LIN {X 0,Y 316.561,Z 503.563,A -85,B 0,C 180,E1 -16116.935,E2 -16116.935} C_VEL
LIN {X 0,Y 317.604,Z 489.042,A -85,B 0,C 180,E1 -16117.711,E2 -16117.711} C_VEL
LIN {X 0,Y 318.34,Z 474.612,A -85,B 0,C 180,E1 -16118.212,E2 -16118.212} C_VEL
LIN {X 0,Y 320.9,Z 379.662,A -85,B 0,C 180,E1 -16120.351,E2 -16120.351} C_VEL
LIN {X 0,Y 312.797,Z 358.488,A -85,B 0,C 180,E1 -16121.547,E2 -16121.547} C_VEL
LIN {X 0,Y 305.815,Z 342.039,A -85,B 0,C 180,E1 -16122.612,E2 -16122.612} C_VEL
LIN {X 0,Y 305.593,Z 341.045,A -85,B 0,C 180,E1 -16122.959,E2 -16122.959} C_VEL
LIN {X 0,Y 305.551,Z 341.05,A -85,B 0,C 180,E1 -16126.023,E2 -16126.023} C_VEL
LIN {X 0,Y 305.541,Z 341.055,A -85,B 0,C 180,E1 -16129.428,E2 -16129.428} C_VEL
LIN {X 0,Y 305.486,Z 341.061,A -85,B 0,C 180,E1 -16133.04,E2 -16133.04} C_VEL
LIN {X 0,Y 305.466,Z 341.058,A -85,B 0,C 180,E1 -16136.197,E2 -16136.197} C_VEL
LIN {X 0,Y 305.433,Z 341.065,A -85,B 0,C 180,E1 -16139.03,E2 -16139.03} C_VEL
LIN {X 0,Y 305.434,Z 341.061,A -85,B 0,C 180,E1 -16141.954,E2 -16141.954} C_VEL
LIN {X 0,Y 305.46,Z 341.058,A -85,B 0,C 180,E1 -16145.115,E2 -16145.115} C_VEL
LIN {X 0,Y 305.432,Z 341.061,A -85,B 0,C 180,E1 -16148.526,E2 -16148.526} C_VEL
LIN {X 0,Y 305.391,Z 341.064,A -85,B 0,C 180,E1 -16149.611,E2 -16149.611} C_VEL
LIN {X 0,Y 304.744,Z 341.152,A -85,B 0,C 180,E1 -16150.712,E2 -16150.712} C_VEL
LIN {X 0,Y 301.909,Z 341.502,A -85,B 0,C 180,E1 -16152.504,E2 -16152.504} C_VEL
LIN {X 0,Y 299.483,Z 341.8,A -85,B 0,C 180,E1 -16153.957,E2 -16153.957} C_VEL
LIN {X 0,Y 298.425,Z 341.93,A -85,B 0,C 180,E1 -16155.083,E2 -16155.083} C_VEL
LIN {X 0,Y 298.331,Z 341.939,A -85,B 0,C 180,E1 -16155.464,E2 -16155.464} C_VEL
LIN {X 0,Y 298.348,Z 341.946,A -85,B 0,C 180,E1 -16158.922,E2 -16158.922} C_VEL
LIN {X 0,Y 298.427,Z 341.922,A -85,B 0,C 180,E1 -16163.199,E2 -16163.199} C_VEL
LIN {X 0,Y 298.394,Z 341.937,A -85,B 0,C 180,E1 -16167.2,E2 -16167.2} C_VEL
LIN {X 0,Y 298.366,Z 341.944,A -85,B 0,C 180,E1 -16170.639,E2 -16170.639} C_VEL
LIN {X 0,Y 298.414,Z 341.937,A -85,B 0,C 180,E1 -16174.918,E2 -16174.918} C_VEL
LIN {X 0,Y 298.394,Z 341.938,A -85,B 0,C 180,E1 -16177.862,E2 -16177.862} C_VEL
LIN {X 0,Y 298.464,Z 341.931,A -85,B 0,C 180,E1 -16180.752,E2 -16180.752} C_VEL
LIN {X 0,Y 298.513,Z 341.917,A -85,B 0,C 180,E1 -16184.991,E2 -16184.991} C_VEL
LIN {X 0,Y 298.585,Z 341.905,A -85,B 0,C 180,E1 -16189.147,E2 -16189.147} C_VEL
LIN {X 0,Y 298.702,Z 341.9,A -85,B 0,C 180,E1 -16191.885,E2 -16191.885} C_VEL
LIN {X 0,Y 298.639,Z 341.908,A -85,B 0,C 180,E1 -16194.599,E2 -16194.599} C_VEL
LIN {X 0,Y 298.92,Z 341.861,A -85,B 0,C 180,E1 -16198.653,E2 -16198.653} C_VEL
LIN {X 0,Y 298.92,Z 341.864,A -85,B 0,C 180,E1 -16201.348,E2 -16201.348} C_VEL
LIN {X 0,Y 298.752,Z 341.893,A -85,B 0,C 180,E1 -16206.755,E2 -16206.755} C_VEL
LIN {X 0,Y 298.63,Z 341.909,A -85,B 0,C 180,E1 -16209.483,E2 -16209.483} C_VEL
LIN {X 0,Y 298.557,Z 341.92,A -85,B 0,C 180,E1 -16213.616,E2 -16213.616} C_VEL
LIN {X 0,Y 298.554,Z 341.919,A -85,B 0,C 180,E1 -16216.409,E2 -16216.409} C_VEL
LIN {X 0,Y 298.516,Z 341.923,A -85,B 0,C 180,E1 -16219.655,E2 -16219.655} C_VEL
LIN {X 0,Y 298.463,Z 341.932,A -85,B 0,C 180,E1 -16223.598,E2 -16223.598} C_VEL
LIN {X 0,Y 298.492,Z 341.925,A -85,B 0,C 180,E1 -16226.575,E2 -16226.575} C_VEL
LIN {X 0,Y 298.421,Z 341.936,A -85,B 0,C 180,E1 -16229.641,E2 -16229.641} C_VEL
LIN {X 0,Y 298.4,Z 341.938,A -85,B 0,C 180,E1 -16232.8,E2 -16232.8} C_VEL
LIN {X 0,Y 298.45,Z 341.932,A -85,B 0,C 180,E1 -16236.807,E2 -16236.807} C_VEL
LIN {X 0,Y 298.393,Z 341.943,A -85,B 0,C 180,E1 -16241.088,E2 -16241.088} C_VEL
LIN {X 0,Y 298.393,Z 341.942,A -85,B 0,C 180,E1 -16245.041,E2 -16245.041} C_VEL
LIN {X 0,Y 298.393,Z 341.944,A -85,B 0,C 180,E1 -16248.912,E2 -16248.912} C_VEL
LIN {X 0,Y 298.451,Z 341.937,A -85,B 0,C 180,E1 -16253.192,E2 -16253.192} C_VEL
LIN {X 0,Y 298.484,Z 342.254,A -85,B 0,C 180,E1 -16253.458,E2 -16253.458} C_VEL
LIN {X 0,Y 301.039,Z 352.934,A -85,B 0,C 180,E1 -16256.6,E2 -16256.6} C_VEL
LIN {X 0,Y 303.03,Z 362.138,A -85,B 0,C 180,E1 -16259.159,E2 -16259.159} C_VEL
LIN {X 0,Y 308.535,Z 376.907,A -85,B 0,C 180,E1 -16260.032,E2 -16260.032} C_VEL
LIN {X 0,Y 313.753,Z 411.636,A -85,B 0,C 180,E1 -16261.349,E2 -16261.349} C_VEL
LIN {X 0,Y 311.27,Z 499.633,A -85,B 0,C 180,E1 -16263.381,E2 -16263.381} C_VEL
LIN {X 0,Y 310.406,Z 513.885,A -85,B 0,C 180,E1 -16263.934,E2 -16263.934} C_VEL
LIN {X 0,Y 309.038,Z 528.229,A -85,B 0,C 180,E1 -16264.759,E2 -16264.759} C_VEL
LIN {X 0,Y 307.585,Z 540.599,A -85,B 0,C 180,E1 -16265.714,E2 -16265.714} C_VEL
LIN {X 0,Y 305.986,Z 553.621,A -85,B 0,C 180,E1 -16267.016,E2 -16267.016} C_VEL
LIN {X 0,Y 304.401,Z 564.227,A -85,B 0,C 180,E1 -16268.32,E2 -16268.32} C_VEL
LIN {X 0,Y 302.566,Z 575.211,A -85,B 0,C 180,E1 -16269.963,E2 -16269.963} C_VEL
LIN {X 0,Y 300.847,Z 586.07,A -85,B 0,C 180,E1 -16271.968,E2 -16271.968} C_VEL
LIN {X 0,Y 299.37,Z 595.713,A -85,B 0,C 180,E1 -16274.162,E2 -16274.162} C_VEL
LIN {X 0,Y 298.435,Z 602.452,A -85,B 0,C 180,E1 -16276.031,E2 -16276.031} C_VEL
LIN {X 0,Y 297.468,Z 609.537,A -85,B 0,C 180,E1 -16278.414,E2 -16278.414} C_VEL
LIN {X 0,Y 296.971,Z 614.436,A -85,B 0,C 180,E1 -16280.463,E2 -16280.463} C_VEL
LIN {X 0,Y 296.656,Z 619.479,A -85,B 0,C 180,E1 -16283.196,E2 -16283.196} C_VEL
LIN {X 0,Y 296.569,Z 622.979,A -85,B 0,C 180,E1 -16285.922,E2 -16285.922} C_VEL
LIN {X 0,Y 296.561,Z 625.044,A -85,B 0,C 180,E1 -16288.641,E2 -16288.641} C_VEL
LIN {X 0,Y 296.583,Z 625.56,A -85,B 0,C 180,E1 -16289.999,E2 -16289.999} C_VEL
LIN {X 0,Y 296.544,Z 625.573,A -85,B 0,C 180,E1 -16292.716,E2 -16292.716} C_VEL
LIN {X 0,Y 296.546,Z 624.19,A -85,B 0,C 180,E1 -16295.507,E2 -16295.507} C_VEL
LIN {X 0,Y 296.813,Z 621.558,A -85,B 0,C 180,E1 -16298.166,E2 -16298.166} C_VEL
LIN {X 0,Y 297.411,Z 617.457,A -85,B 0,C 180,E1 -16300.896,E2 -16300.896} C_VEL
LIN {X 0,Y 298.62,Z 611.832,A -85,B 0,C 180,E1 -16303.611,E2 -16303.611} C_VEL
LIN {X 0,Y 300.197,Z 604.52,A -85,B 0,C 180,E1 -16306.315,E2 -16306.315} C_VEL
LIN {X 0,Y 302.199,Z 596.494,A -85,B 0,C 180,E1 -16308.648,E2 -16308.648} C_VEL
LIN {X 0,Y 304.312,Z 588.131,A -85,B 0,C 180,E1 -16310.62,E2 -16310.62} C_VEL
LIN {X 0,Y 306.857,Z 578.101,A -85,B 0,C 180,E1 -16312.557,E2 -16312.557} C_VEL
LIN {X 0,Y 309.221,Z 568.042,A -85,B 0,C 180,E1 -16314.147,E2 -16314.147} C_VEL
LIN {X 0,Y 311.767,Z 555.927,A -85,B 0,C 180,E1 -16315.716,E2 -16315.716} C_VEL
LIN {X 0,Y 314.08,Z 543.986,A -85,B 0,C 180,E1 -16316.943,E2 -16316.943} C_VEL
LIN {X 0,Y 316.223,Z 530.835,A -85,B 0,C 180,E1 -16318,E2 -16318} C_VEL
LIN {X 0,Y 318.041,Z 517.262,A -85,B 0,C 180,E1 -16318.815,E2 -16318.815} C_VEL
LIN {X 0,Y 319.406,Z 503.345,A -85,B 0,C 180,E1 -16319.401,E2 -16319.401} C_VEL
LIN {X 0,Y 320.305,Z 484.536,A -85,B 0,C 180,E1 -16319.898,E2 -16319.898} C_VEL
LIN {X 0,Y 322.883,Z 413.283,A -85,B 0,C 180,E1 -16321.53,E2 -16321.53} C_VEL
LIN {X 0,Y 320.316,Z 397.518,A -85,B 0,C 180,E1 -16322.31,E2 -16322.31} C_VEL
LIN {X 0,Y 318.901,Z 390.848,A -85,B 0,C 180,E1 -16322.692,E2 -16322.692} C_VEL
LIN {X 0,Y 312.51,Z 377.162,A -85,B 0,C 180,E1 -16324.007,E2 -16324.007} C_VEL
LIN {X 0,Y 306.262,Z 365.122,A -85,B 0,C 180,E1 -16325.339,E2 -16325.339} C_VEL
LIN {X 0,Y 303.755,Z 360.397,A -85,B 0,C 180,E1 -16325.923,E2 -16325.923} C_VEL
LIN {X 0,Y 300.958,Z 350.238,A -85,B 0,C 180,E1 -16329.59,E2 -16329.59} C_VEL
LIN {X 0,Y 298.426,Z 341.929,A -85,B 0,C 180,E1 -16332.924,E2 -16332.924} C_VEL
LIN {X 0,Y 298.398,Z 341.929,A -85,B 0,C 180,E1 -16336.919,E2 -16336.919} C_VEL
LIN {X 0,Y 298.41,Z 341.919,A -85,B 0,C 180,E1 -16341.002,E2 -16341.002} C_VEL
LIN {X 0,Y 298.426,Z 341.933,A -85,B 0,C 180,E1 -16343.931,E2 -16343.931} C_VEL
LIN {X 0,Y 298.39,Z 341.937,A -85,B 0,C 180,E1 -16347.982,E2 -16347.982} C_VEL
LIN {X 0,Y 298.458,Z 341.933,A -85,B 0,C 180,E1 -16351.903,E2 -16351.903} C_VEL
LIN {X 0,Y 298.479,Z 341.931,A -85,B 0,C 180,E1 -16354.923,E2 -16354.923} C_VEL
LIN {X 0,Y 298.443,Z 341.935,A -85,B 0,C 180,E1 -16359.314,E2 -16359.314} C_VEL
LIN {X 0,Y 298.531,Z 341.92,A -85,B 0,C 180,E1 -16362.179,E2 -16362.179} C_VEL
LIN {X 0,Y 298.586,Z 341.906,A -85,B 0,C 180,E1 -16364.994,E2 -16364.994} C_VEL
LIN {X 0,Y 298.586,Z 341.905,A -85,B 0,C 180,E1 -16369.146,E2 -16369.146} C_VEL
LIN {X 0,Y 298.75,Z 341.892,A -85,B 0,C 180,E1 -16371.885,E2 -16371.885} C_VEL
LIN {X 0,Y 298.643,Z 341.909,A -85,B 0,C 180,E1 -16374.598,E2 -16374.598} C_VEL
LIN {X 0,Y 298.906,Z 341.876,A -85,B 0,C 180,E1 -16378.652,E2 -16378.652} C_VEL
LIN {X 0,Y 298.895,Z 341.869,A -85,B 0,C 180,E1 -16381.347,E2 -16381.347} C_VEL
LIN {X 0,Y 298.693,Z 341.9,A -85,B 0,C 180,E1 -16386.513,E2 -16386.513} C_VEL
LIN {X 0,Y 298.616,Z 341.905,A -85,B 0,C 180,E1 -16389.482,E2 -16389.482} C_VEL
LIN {X 0,Y 298.534,Z 341.919,A -85,B 0,C 180,E1 -16393.616,E2 -16393.616} C_VEL
LIN {X 0,Y 298.474,Z 341.923,A -85,B 0,C 180,E1 -16396.412,E2 -16396.412} C_VEL
LIN {X 0,Y 298.451,Z 341.929,A -85,B 0,C 180,E1 -16399.627,E2 -16399.627} C_VEL
LIN {X 0,Y 298.411,Z 341.941,A -85,B 0,C 180,E1 -16403.601,E2 -16403.601} C_VEL
LIN {X 0,Y 298.399,Z 341.943,A -85,B 0,C 180,E1 -16406.582,E2 -16406.582} C_VEL
LIN {X 0,Y 298.385,Z 341.93,A -85,B 0,C 180,E1 -16409.644,E2 -16409.644} C_VEL
LIN {X 0,Y 298.384,Z 341.932,A -85,B 0,C 180,E1 -16412.801,E2 -16412.801} C_VEL
LIN {X 0,Y 298.448,Z 342.109,A -85,B 0,C 180,E1 -16414.496,E2 -16414.496} C_VEL
LIN {X 0,Y 299.073,Z 344.176,A -85,B 0,C 180,E1 -16415.356,E2 -16415.356} C_VEL
LIN {X 0,Y 301.615,Z 348.304,A -85,B 0,C 180,E1 -16415.931,E2 -16415.931} C_VEL
LIN {X 0,Y 309.75,Z 361.63,A -85,B 0,C 180,E1 -16417.672,E2 -16417.672} C_VEL
LIN {X 0,Y 318.436,Z 377.963,A -85,B 0,C 180,E1 -16419.442,E2 -16419.442} C_VEL
LIN {X 0,Y 323.82,Z 389.532,A -85,B 0,C 180,E1 -16420.501,E2 -16420.501} C_VEL
LIN {X 0,Y 320.298,Z 479.035,A -85,B 0,C 180,E1 -16422.55,E2 -16422.55} C_VEL
LIN {X 0,Y 319.269,Z 493.289,A -85,B 0,C 180,E1 -16423.111,E2 -16423.111} C_VEL
LIN {X 0,Y 317.836,Z 506.14,A -85,B 0,C 180,E1 -16423.832,E2 -16423.832} C_VEL
LIN {X 0,Y 316.098,Z 519.195,A -85,B 0,C 180,E1 -16424.828,E2 -16424.828} C_VEL
LIN {X 0,Y 313.944,Z 531.813,A -85,B 0,C 180,E1 -16426.057,E2 -16426.057} C_VEL
LIN {X 0,Y 311.486,Z 544.174,A -85,B 0,C 180,E1 -16427.577,E2 -16427.577} C_VEL
LIN {X 0,Y 308.852,Z 555.794,A -85,B 0,C 180,E1 -16429.357,E2 -16429.357} C_VEL
LIN {X 0,Y 306.313,Z 566.384,A -85,B 0,C 180,E1 -16431.383,E2 -16431.383} C_VEL
LIN {X 0,Y 304.021,Z 575.007,A -85,B 0,C 180,E1 -16433.415,E2 -16433.415} C_VEL
LIN {X 0,Y 301.963,Z 582.651,A -85,B 0,C 180,E1 -16435.641,E2 -16435.641} C_VEL
LIN {X 0,Y 300.116,Z 589.603,A -85,B 0,C 180,E1 -16438.206,E2 -16438.206} C_VEL
LIN {X 0,Y 298.826,Z 594.434,A -85,B 0,C 180,E1 -16440.48,E2 -16440.48} C_VEL
LIN {X 0,Y 297.685,Z 598.912,A -85,B 0,C 180,E1 -16443.35,E2 -16443.35} C_VEL
LIN {X 0,Y 296.885,Z 601.861,A -85,B 0,C 180,E1 -16446.271,E2 -16446.271} C_VEL
LIN {X 0,Y 296.685,Z 602.753,A -85,B 0,C 180,E1 -16447.729,E2 -16447.729} C_VEL
LIN {X 0,Y 296.391,Z 603.41,A -85,B 0,C 180,E1 -16450.613,E2 -16450.613} C_VEL
LIN {X 0,Y 296.359,Z 603.175,A -85,B 0,C 180,E1 -16452.045,E2 -16452.045} C_VEL
LIN {X 0,Y 296.359,Z 601.642,A -85,B 0,C 180,E1 -16454.88,E2 -16454.88} C_VEL
LIN {X 0,Y 296.559,Z 600.305,A -85,B 0,C 180,E1 -16456.319,E2 -16456.319} C_VEL
LIN {X 0,Y 296.964,Z 596.634,A -85,B 0,C 180,E1 -16459.088,E2 -16459.088} C_VEL
LIN {X 0,Y 297.636,Z 591.401,A -85,B 0,C 180,E1 -16461.856,E2 -16461.856} C_VEL
LIN {X 0,Y 298.375,Z 586.318,A -85,B 0,C 180,E1 -16463.917,E2 -16463.917} C_VEL
LIN {X 0,Y 299.441,Z 579.063,A -85,B 0,C 180,E1 -16466.301,E2 -16466.301} C_VEL
LIN {X 0,Y 300.707,Z 571.447,A -85,B 0,C 180,E1 -16468.327,E2 -16468.327} C_VEL
LIN {X 0,Y 302.204,Z 562.576,A -85,B 0,C 180,E1 -16470.278,E2 -16470.278} C_VEL
LIN {X 0,Y 303.619,Z 553.219,A -85,B 0,C 180,E1 -16471.991,E2 -16471.991} C_VEL
LIN {X 0,Y 305.369,Z 542.327,A -85,B 0,C 180,E1 -16473.63,E2 -16473.63} C_VEL
LIN {X 0,Y 307.014,Z 530.442,A -85,B 0,C 180,E1 -16475.09,E2 -16475.09} C_VEL
LIN {X 0,Y 308.604,Z 517.319,A -85,B 0,C 180,E1 -16476.375,E2 -16476.375} C_VEL
LIN {X 0,Y 309.972,Z 503.451,A -85,B 0,C 180,E1 -16477.41,E2 -16477.41} C_VEL
LIN {X 0,Y 311.041,Z 488.778,A -85,B 0,C 180,E1 -16478.201,E2 -16478.201} C_VEL
LIN {X 0,Y 311.728,Z 475.513,A -85,B 0,C 180,E1 -16478.673,E2 -16478.673} C_VEL
LIN {X 0,Y 314.484,Z 381.922,A -85,B 0,C 180,E1 -16480.813,E2 -16480.813} C_VEL
LIN {X 0,Y 308.384,Z 365.374,A -85,B 0,C 180,E1 -16481.754,E2 -16481.754} C_VEL
LIN {X 0,Y 299.779,Z 345.144,A -85,B 0,C 180,E1 -16483.072,E2 -16483.072} C_VEL
LIN {X 0,Y 298.606,Z 342.346,A -85,B 0,C 180,E1 -16483.268,E2 -16483.268} C_VEL
LIN {X 0,Y 298.552,Z 341.923,A -85,B 0,C 180,E1 -16483.443,E2 -16483.443} C_VEL
LIN {X 0,Y 298.485,Z 341.931,A -85,B 0,C 180,E1 -16486.413,E2 -16486.413} C_VEL
LIN {X 0,Y 298.482,Z 341.933,A -85,B 0,C 180,E1 -16489.64,E2 -16489.64} C_VEL
LIN {X 0,Y 298.419,Z 341.938,A -85,B 0,C 180,E1 -16493.602,E2 -16493.602} C_VEL
LIN {X 0,Y 298.406,Z 341.939,A -85,B 0,C 180,E1 -16496.583,E2 -16496.583} C_VEL
LIN {X 0,Y 298.36,Z 341.944,A -85,B 0,C 180,E1 -16499.649,E2 -16499.649} C_VEL
LIN {X 0,Y 298.391,Z 341.942,A -85,B 0,C 180,E1 -16502.802,E2 -16502.802} C_VEL
LIN {X 0,Y 298.427,Z 341.931,A -85,B 0,C 180,E1 -16506.803,E2 -16506.803} C_VEL
LIN {X 0,Y 298.365,Z 341.942,A -85,B 0,C 180,E1 -16509.591,E2 -16509.591} C_VEL
LIN {X 0,Y 298.369,Z 341.936,A -85,B 0,C 180,E1 -16513.098,E2 -16513.098} C_VEL
LIN {X 0,Y 298.331,Z 341.939,A -85,B 0,C 180,E1 -16515.464,E2 -16515.464} C_VEL
LIN {X 0,Y 297.645,Z 342.031,A -85,B 0,C 180,E1 -16516.592,E2 -16516.592} C_VEL
LIN {X 0,Y 294.807,Z 342.387,A -85,B 0,C 180,E1 -16518.429,E2 -16518.429} C_VEL
LIN {X 0,Y 292.411,Z 342.685,A -85,B 0,C 180,E1 -16519.919,E2 -16519.919} C_VEL
LIN {X 0,Y 291.383,Z 342.808,A -85,B 0,C 180,E1 -16521.073,E2 -16521.073} C_VEL
LIN {X 0,Y 291.298,Z 342.815,A -85,B 0,C 180,E1 -16521.463,E2 -16521.463} C_VEL
LIN {X 0,Y 291.356,Z 342.804,A -85,B 0,C 180,E1 -16524.626,E2 -16524.626} C_VEL
LIN {X 0,Y 291.367,Z 342.812,A -85,B 0,C 180,E1 -16527.951,E2 -16527.951} C_VEL
LIN {X 0,Y 291.317,Z 342.818,A -85,B 0,C 180,E1 -16531.152,E2 -16531.152} C_VEL
LIN {X 0,Y 291.344,Z 342.819,A -85,B 0,C 180,E1 -16534.266,E2 -16534.266} C_VEL
LIN {X 0,Y 291.352,Z 342.813,A -85,B 0,C 180,E1 -16537.298,E2 -16537.298} C_VEL
LIN {X 0,Y 291.389,Z 342.813,A -85,B 0,C 180,E1 -16540.266,E2 -16540.266} C_VEL
LIN {X 0,Y 291.477,Z 342.794,A -85,B 0,C 180,E1 -16544.683,E2 -16544.683} C_VEL
LIN {X 0,Y 291.531,Z 342.784,A -85,B 0,C 180,E1 -16548.881,E2 -16548.881} C_VEL
LIN {X 0,Y 291.655,Z 342.776,A -85,B 0,C 180,E1 -16551.687,E2 -16551.687} C_VEL
LIN {X 0,Y 291.608,Z 342.784,A -85,B 0,C 180,E1 -16554.468,E2 -16554.468} C_VEL
LIN {X 0,Y 291.886,Z 342.735,A -85,B 0,C 180,E1 -16558.621,E2 -16558.621} C_VEL
LIN {X 0,Y 291.886,Z 342.739,A -85,B 0,C 180,E1 -16561.38,E2 -16561.38} C_VEL
LIN {X 0,Y 291.704,Z 342.771,A -85,B 0,C 180,E1 -16566.919,E2 -16566.919} C_VEL
LIN {X 0,Y 291.573,Z 342.789,A -85,B 0,C 180,E1 -16569.714,E2 -16569.714} C_VEL
LIN {X 0,Y 291.527,Z 342.795,A -85,B 0,C 180,E1 -16573.95,E2 -16573.95} C_VEL
LIN {X 0,Y 291.492,Z 342.798,A -85,B 0,C 180,E1 -16576.818,E2 -16576.818} C_VEL
LIN {X 0,Y 291.456,Z 342.802,A -85,B 0,C 180,E1 -16579.875,E2 -16579.875} C_VEL
LIN {X 0,Y 291.405,Z 342.806,A -85,B 0,C 180,E1 -16584.205,E2 -16584.205} C_VEL
LIN {X 0,Y 291.425,Z 342.808,A -85,B 0,C 180,E1 -16587.272,E2 -16587.272} C_VEL
LIN {X 0,Y 291.339,Z 342.816,A -85,B 0,C 180,E1 -16590.437,E2 -16590.437} C_VEL
LIN {X 0,Y 291.349,Z 342.818,A -85,B 0,C 180,E1 -16593.698,E2 -16593.698} C_VEL
LIN {X 0,Y 291.378,Z 342.811,A -85,B 0,C 180,E1 -16597.253,E2 -16597.253} C_VEL
LIN {X 0,Y 291.338,Z 342.819,A -85,B 0,C 180,E1 -16600.642,E2 -16600.642} C_VEL
LIN {X 0,Y 291.319,Z 342.82,A -85,B 0,C 180,E1 -16604.397,E2 -16604.397} C_VEL
LIN {X 0,Y 291.332,Z 342.821,A -85,B 0,C 180,E1 -16608.404,E2 -16608.404} C_VEL
LIN {X 0,Y 291.358,Z 342.823,A -85,B 0,C 180,E1 -16611.158,E2 -16611.158} C_VEL
LIN {X 0,Y 291.416,Z 342.879,A -85,B 0,C 180,E1 -16612.864,E2 -16612.864} C_VEL
LIN {X 0,Y 294.4,Z 355.607,A -85,B 0,C 180,E1 -16616.696,E2 -16616.696} C_VEL
LIN {X 0,Y 295.8,Z 362.018,A -85,B 0,C 180,E1 -16618.485,E2 -16618.485} C_VEL
LIN {X 0,Y 302.3,Z 379.135,A -85,B 0,C 180,E1 -16619.54,E2 -16619.54} C_VEL
LIN {X 0,Y 307.271,Z 412.118,A -85,B 0,C 180,E1 -16620.83,E2 -16620.83} C_VEL
LIN {X 0,Y 304.68,Z 499.831,A -85,B 0,C 180,E1 -16622.897,E2 -16622.897} C_VEL
LIN {X 0,Y 303.777,Z 513.874,A -85,B 0,C 180,E1 -16623.46,E2 -16623.46} C_VEL
LIN {X 0,Y 302.45,Z 527.587,A -85,B 0,C 180,E1 -16624.262,E2 -16624.262} C_VEL
LIN {X 0,Y 300.833,Z 540.883,A -85,B 0,C 180,E1 -16625.311,E2 -16625.311} C_VEL
LIN {X 0,Y 299.184,Z 553.839,A -85,B 0,C 180,E1 -16626.645,E2 -16626.645} C_VEL
LIN {X 0,Y 297.548,Z 564.359,A -85,B 0,C 180,E1 -16627.977,E2 -16627.977} C_VEL
LIN {X 0,Y 295.81,Z 574.283,A -85,B 0,C 180,E1 -16629.485,E2 -16629.485} C_VEL
LIN {X 0,Y 294.309,Z 583.605,A -85,B 0,C 180,E1 -16631.192,E2 -16631.192} C_VEL
LIN {X 0,Y 292.8,Z 592.929,A -85,B 0,C 180,E1 -16633.259,E2 -16633.259} C_VEL
LIN {X 0,Y 291.727,Z 600.692,A -85,B 0,C 180,E1 -16635.346,E2 -16635.346} C_VEL
LIN {X 0,Y 290.735,Z 607.131,A -85,B 0,C 180,E1 -16637.433,E2 -16637.433} C_VEL
LIN {X 0,Y 290.044,Z 612.404,A -85,B 0,C 180,E1 -16639.528,E2 -16639.528} C_VEL
LIN {X 0,Y 289.648,Z 617.954,A -85,B 0,C 180,E1 -16642.33,E2 -16642.33} C_VEL
LIN {X 0,Y 289.482,Z 621.101,A -85,B 0,C 180,E1 -16644.5,E2 -16644.5} C_VEL
LIN {X 0,Y 289.496,Z 623.832,A -85,B 0,C 180,E1 -16647.216,E2 -16647.216} C_VEL
LIN {X 0,Y 289.498,Z 625.253,A -85,B 0,C 180,E1 -16649.999,E2 -16649.999} C_VEL
LIN {X 0,Y 289.469,Z 625.316,A -85,B 0,C 180,E1 -16652.782,E2 -16652.782} C_VEL
LIN {X 0,Y 289.477,Z 624.043,A -85,B 0,C 180,E1 -16655.572,E2 -16655.572} C_VEL
LIN {X 0,Y 289.746,Z 621.425,A -85,B 0,C 180,E1 -16658.367,E2 -16658.367} C_VEL
LIN {X 0,Y 290.377,Z 617.387,A -85,B 0,C 180,E1 -16661.163,E2 -16661.163} C_VEL
LIN {X 0,Y 291.695,Z 611.822,A -85,B 0,C 180,E1 -16663.94,E2 -16663.94} C_VEL
LIN {X 0,Y 293.21,Z 605.153,A -85,B 0,C 180,E1 -16666.509,E2 -16666.509} C_VEL
LIN {X 0,Y 295.119,Z 597.853,A -85,B 0,C 180,E1 -16668.752,E2 -16668.752} C_VEL
LIN {X 0,Y 297.678,Z 588.348,A -85,B 0,C 180,E1 -16671.101,E2 -16671.101} C_VEL
LIN {X 0,Y 300.323,Z 578.429,A -85,B 0,C 180,E1 -16673.076,E2 -16673.076} C_VEL
LIN {X 0,Y 303.167,Z 567.022,A -85,B 0,C 180,E1 -16674.915,E2 -16674.915} C_VEL
LIN {X 0,Y 305.744,Z 555.232,A -85,B 0,C 180,E1 -16676.445,E2 -16676.445} C_VEL
LIN {X 0,Y 308.101,Z 543.195,A -85,B 0,C 180,E1 -16677.694,E2 -16677.694} C_VEL
LIN {X 0,Y 310.375,Z 529.89,A -85,B 0,C 180,E1 -16678.761,E2 -16678.761} C_VEL
LIN {X 0,Y 312.328,Z 515.344,A -85,B 0,C 180,E1 -16679.625,E2 -16679.625} C_VEL
LIN {X 0,Y 313.773,Z 500.621,A -85,B 0,C 180,E1 -16680.215,E2 -16680.215} C_VEL
LIN {X 0,Y 314.992,Z 472.314,A -85,B 0,C 180,E1 -16680.91,E2 -16680.91} C_VEL
LIN {X 0,Y 317.16,Z 414.775,A -85,B 0,C 180,E1 -16682.25,E2 -16682.25} C_VEL
LIN {X 0,Y 314.703,Z 399.1,A -85,B 0,C 180,E1 -16683.043,E2 -16683.043} C_VEL
LIN {X 0,Y 313.498,Z 393.641,A -85,B 0,C 180,E1 -16683.376,E2 -16683.376} C_VEL
LIN {X 0,Y 306.099,Z 377.891,A -85,B 0,C 180,E1 -16684.969,E2 -16684.969} C_VEL
LIN {X 0,Y 301.082,Z 368.602,A -85,B 0,C 180,E1 -16686.076,E2 -16686.076} C_VEL
LIN {X 0,Y 298.386,Z 363.841,A -85,B 0,C 180,E1 -16686.688,E2 -16686.688} C_VEL
LIN {X 0,Y 296.483,Z 360.11,A -85,B 0,C 180,E1 -16687.149,E2 -16687.149} C_VEL
LIN {X 0,Y 293.87,Z 351.045,A -85,B 0,C 180,E1 -16690.605,E2 -16690.605} C_VEL
LIN {X 0,Y 291.526,Z 343.737,A -85,B 0,C 180,E1 -16693.678,E2 -16693.678} C_VEL
LIN {X 0,Y 291.328,Z 342.822,A -85,B 0,C 180,E1 -16694.079,E2 -16694.079} C_VEL
LIN {X 0,Y 291.322,Z 342.82,A -85,B 0,C 180,E1 -16698.403,E2 -16698.403} C_VEL
LIN {X 0,Y 291.36,Z 342.798,A -85,B 0,C 180,E1 -16701.159,E2 -16701.159} C_VEL
LIN {X 0,Y 291.38,Z 342.81,A -85,B 0,C 180,E1 -16704.628,E2 -16704.628} C_VEL
LIN {X 0,Y 291.367,Z 342.812,A -85,B 0,C 180,E1 -16707.95,E2 -16707.95} C_VEL
LIN {X 0,Y 291.377,Z 342.812,A -85,B 0,C 180,E1 -16711.157,E2 -16711.157} C_VEL
LIN {X 0,Y 291.41,Z 342.804,A -85,B 0,C 180,E1 -16714.271,E2 -16714.271} C_VEL
LIN {X 0,Y 291.374,Z 342.805,A -85,B 0,C 180,E1 -16717.298,E2 -16717.298} C_VEL
LIN {X 0,Y 291.451,Z 342.798,A -85,B 0,C 180,E1 -16720.269,E2 -16720.269} C_VEL
LIN {X 0,Y 291.548,Z 342.783,A -85,B 0,C 180,E1 -16724.623,E2 -16724.623} C_VEL
LIN {X 0,Y 291.529,Z 342.784,A -85,B 0,C 180,E1 -16728.88,E2 -16728.88} C_VEL
LIN {X 0,Y 291.701,Z 342.772,A -85,B 0,C 180,E1 -16731.688,E2 -16731.688} C_VEL
LIN {X 0,Y 291.615,Z 342.784,A -85,B 0,C 180,E1 -16734.468,E2 -16734.468} C_VEL
LIN {X 0,Y 291.872,Z 342.752,A -85,B 0,C 180,E1 -16738.62,E2 -16738.62} C_VEL
LIN {X 0,Y 291.863,Z 342.744,A -85,B 0,C 180,E1 -16741.379,E2 -16741.379} C_VEL
LIN {X 0,Y 291.675,Z 342.777,A -85,B 0,C 180,E1 -16746.919,E2 -16746.919} C_VEL
LIN {X 0,Y 291.559,Z 342.786,A -85,B 0,C 180,E1 -16749.714,E2 -16749.714} C_VEL
LIN {X 0,Y 291.505,Z 342.798,A -85,B 0,C 180,E1 -16753.951,E2 -16753.951} C_VEL
LIN {X 0,Y 291.419,Z 342.804,A -85,B 0,C 180,E1 -16756.821,E2 -16756.821} C_VEL
LIN {X 0,Y 291.415,Z 342.806,A -85,B 0,C 180,E1 -16759.86,E2 -16759.86} C_VEL
LIN {X 0,Y 291.351,Z 342.818,A -85,B 0,C 180,E1 -16764.209,E2 -16764.209} C_VEL
LIN {X 0,Y 291.344,Z 342.811,A -85,B 0,C 180,E1 -16767.279,E2 -16767.279} C_VEL
LIN {X 0,Y 291.31,Z 342.823,A -85,B 0,C 180,E1 -16770.439,E2 -16770.439} C_VEL
LIN {X 0,Y 291.337,Z 342.864,A -85,B 0,C 180,E1 -16773.306,E2 -16773.306} C_VEL
LIN {X 0,Y 291.825,Z 344.645,A -85,B 0,C 180,E1 -16774.037,E2 -16774.037} C_VEL
LIN {X 0,Y 298.875,Z 355.611,A -85,B 0,C 180,E1 -16775.694,E2 -16775.694} C_VEL
LIN {X 0,Y 306.082,Z 367.778,A -85,B 0,C 180,E1 -16777.283,E2 -16777.283} C_VEL
LIN {X 0,Y 313.892,Z 382.695,A -85,B 0,C 180,E1 -16778.925,E2 -16778.925} C_VEL
LIN {X 0,Y 317.955,Z 391.51,A -85,B 0,C 180,E1 -16779.763,E2 -16779.763} C_VEL
LIN {X 0,Y 314.989,Z 467.229,A -85,B 0,C 180,E1 -16781.513,E2 -16781.513} C_VEL
LIN {X 0,Y 314.15,Z 483.905,A -85,B 0,C 180,E1 -16781.976,E2 -16781.976} C_VEL
LIN {X 0,Y 312.894,Z 498.513,A -85,B 0,C 180,E1 -16782.644,E2 -16782.644} C_VEL
LIN {X 0,Y 311.214,Z 511.756,A -85,B 0,C 180,E1 -16783.495,E2 -16783.495} C_VEL
LIN {X 0,Y 309.384,Z 523.994,A -85,B 0,C 180,E1 -16784.541,E2 -16784.541} C_VEL
LIN {X 0,Y 306.898,Z 536.881,A -85,B 0,C 180,E1 -16785.928,E2 -16785.928} C_VEL
LIN {X 0,Y 304.284,Z 548.792,A -85,B 0,C 180,E1 -16787.548,E2 -16787.548} C_VEL
LIN {X 0,Y 301.743,Z 559.208,A -85,B 0,C 180,E1 -16789.298,E2 -16789.298} C_VEL
LIN {X 0,Y 299.461,Z 568.078,A -85,B 0,C 180,E1 -16791.115,E2 -16791.115} C_VEL
LIN {X 0,Y 296.964,Z 577.007,A -85,B 0,C 180,E1 -16793.348,E2 -16793.348} C_VEL
LIN {X 0,Y 294.954,Z 584.071,A -85,B 0,C 180,E1 -16795.537,E2 -16795.537} C_VEL
LIN {X 0,Y 293.037,Z 590.787,A -85,B 0,C 180,E1 -16798.156,E2 -16798.156} C_VEL
LIN {X 0,Y 291.95,Z 594.674,A -85,B 0,C 180,E1 -16800.066,E2 -16800.066} C_VEL
LIN {X 0,Y 290.844,Z 598.747,A -85,B 0,C 180,E1 -16802.671,E2 -16802.671} C_VEL
LIN {X 0,Y 289.909,Z 601.862,A -85,B 0,C 180,E1 -16805.664,E2 -16805.664} C_VEL
LIN {X 0,Y 289.447,Z 603.435,A -85,B 0,C 180,E1 -16808.642,E2 -16808.642} C_VEL
LIN {X 0,Y 289.275,Z 603.534,A -85,B 0,C 180,E1 -16811.59,E2 -16811.59} C_VEL
LIN {X 0,Y 289.247,Z 602.188,A -85,B 0,C 180,E1 -16814.499,E2 -16814.499} C_VEL
LIN {X 0,Y 289.576,Z 599.371,A -85,B 0,C 180,E1 -16817.385,E2 -16817.385} C_VEL
LIN {X 0,Y 290.112,Z 595.078,A -85,B 0,C 180,E1 -16820.238,E2 -16820.238} C_VEL
LIN {X 0,Y 290.991,Z 589.186,A -85,B 0,C 180,E1 -16823.065,E2 -16823.065} C_VEL
LIN {X 0,Y 291.94,Z 582.57,A -85,B 0,C 180,E1 -16825.514,E2 -16825.514} C_VEL
LIN {X 0,Y 293.329,Z 574.34,A -85,B 0,C 180,E1 -16827.942,E2 -16827.942} C_VEL
LIN {X 0,Y 294.828,Z 565.718,A -85,B 0,C 180,E1 -16830.001,E2 -16830.001} C_VEL
LIN {X 0,Y 296.481,Z 555.302,A -85,B 0,C 180,E1 -16832.039,E2 -16832.039} C_VEL
LIN {X 0,Y 298.241,Z 544.778,A -85,B 0,C 180,E1 -16833.717,E2 -16833.717} C_VEL
LIN {X 0,Y 299.898,Z 533.362,A -85,B 0,C 180,E1 -16835.211,E2 -16835.211} C_VEL
LIN {X 0,Y 301.536,Z 520.857,A -85,B 0,C 180,E1 -16836.525,E2 -16836.525} C_VEL
LIN {X 0,Y 303.062,Z 506.892,A -85,B 0,C 180,E1 -16837.664,E2 -16837.664} C_VEL
LIN {X 0,Y 304.183,Z 492.857,A -85,B 0,C 180,E1 -16838.513,E2 -16838.513} C_VEL
LIN {X 0,Y 305.046,Z 477.915,A -85,B 0,C 180,E1 -16839.115,E2 -16839.115} C_VEL
LIN {X 0,Y 307.96,Z 383.121,A -85,B 0,C 180,E1 -16841.334,E2 -16841.334} C_VEL
LIN {X 0,Y 300.919,Z 364.584,A -85,B 0,C 180,E1 -16842.447,E2 -16842.447} C_VEL
LIN {X 0,Y 293.875,Z 348.348,A -85,B 0,C 180,E1 -16843.553,E2 -16843.553} C_VEL
LIN {X 0,Y 291.65,Z 343.573,A -85,B 0,C 180,E1 -16843.904,E2 -16843.904} C_VEL
LIN {X 0,Y 291.514,Z 342.799,A -85,B 0,C 180,E1 -16843.952,E2 -16843.952} C_VEL
LIN {X 0,Y 291.438,Z 342.81,A -85,B 0,C 180,E1 -16848.271,E2 -16848.271} C_VEL
LIN {X 0,Y 291.352,Z 342.823,A -85,B 0,C 180,E1 -16851.214,E2 -16851.214} C_VEL
LIN {X 0,Y 291.358,Z 342.816,A -85,B 0,C 180,E1 -16854.21,E2 -16854.21} C_VEL
LIN {X 0,Y 291.35,Z 342.819,A -85,B 0,C 180,E1 -16857.28,E2 -16857.28} C_VEL
LIN {X 0,Y 291.302,Z 342.823,A -85,B 0,C 180,E1 -16860.442,E2 -16860.442} C_VEL
LIN {X 0,Y 291.343,Z 342.818,A -85,B 0,C 180,E1 -16863.7,E2 -16863.7} C_VEL
LIN {X 0,Y 291.358,Z 342.813,A -85,B 0,C 180,E1 -16867.25,E2 -16867.25} C_VEL
LIN {X 0,Y 291.3,Z 342.826,A -85,B 0,C 180,E1 -16870.649,E2 -16870.649} C_VEL
LIN {X 0,Y 291.282,Z 342.816,A -85,B 0,C 180,E1 -16874.405,E2 -16874.405} C_VEL
LIN {X 0,Y 291.295,Z 342.824,A -85,B 0,C 180,E1 -16878.413,E2 -16878.413} C_VEL
LIN {X 0,Y 291.298,Z 342.815,A -85,B 0,C 180,E1 -16881.463,E2 -16881.463} C_VEL
LIN {X 0,Y 290.638,Z 342.896,A -85,B 0,C 180,E1 -16882.618,E2 -16882.618} C_VEL
LIN {X 0,Y 287.827,Z 343.244,A -85,B 0,C 180,E1 -16884.5,E2 -16884.5} C_VEL
LIN {X 0,Y 285.428,Z 343.548,A -85,B 0,C 180,E1 -16886.028,E2 -16886.028} C_VEL
LIN {X 0,Y 284.377,Z 343.683,A -85,B 0,C 180,E1 -16887.21,E2 -16887.21} C_VEL
LIN {X 0,Y 284.28,Z 343.694,A -85,B 0,C 180,E1 -16887.611,E2 -16887.611} C_VEL
LIN {X 0,Y 284.311,Z 343.697,A -85,B 0,C 180,E1 -16890.371,E2 -16890.371} C_VEL
LIN {X 0,Y 284.297,Z 343.693,A -85,B 0,C 180,E1 -16893.579,E2 -16893.579} C_VEL
LIN {X 0,Y 284.31,Z 343.693,A -85,B 0,C 180,E1 -16896.703,E2 -16896.703} C_VEL
LIN {X 0,Y 284.337,Z 343.689,A -85,B 0,C 180,E1 -16899.929,E2 -16899.929} C_VEL
LIN {X 0,Y 284.417,Z 343.674,A -85,B 0,C 180,E1 -16904.517,E2 -16904.517} C_VEL
LIN {X 0,Y 284.462,Z 343.662,A -85,B 0,C 180,E1 -16908.601,E2 -16908.601} C_VEL
LIN {X 0,Y 284.612,Z 343.652,A -85,B 0,C 180,E1 -16911.48,E2 -16911.48} C_VEL
LIN {X 0,Y 284.577,Z 343.661,A -85,B 0,C 180,E1 -16914.331,E2 -16914.331} C_VEL
LIN {X 0,Y 284.853,Z 343.61,A -85,B 0,C 180,E1 -16918.587,E2 -16918.587} C_VEL
LIN {X 0,Y 284.852,Z 343.615,A -85,B 0,C 180,E1 -16921.414,E2 -16921.414} C_VEL
LIN {X 0,Y 284.658,Z 343.649,A -85,B 0,C 180,E1 -16927.092,E2 -16927.092} C_VEL
LIN {X 0,Y 284.519,Z 343.67,A -85,B 0,C 180,E1 -16929.957,E2 -16929.957} C_VEL
LIN {X 0,Y 284.487,Z 343.67,A -85,B 0,C 180,E1 -16934.303,E2 -16934.303} C_VEL
LIN {X 0,Y 284.43,Z 343.679,A -85,B 0,C 180,E1 -16937.248,E2 -16937.248} C_VEL
LIN {X 0,Y 284.385,Z 343.682,A -85,B 0,C 180,E1 -16940.242,E2 -16940.242} C_VEL
LIN {X 0,Y 284.374,Z 343.684,A -85,B 0,C 180,E1 -16943.875,E2 -16943.875} C_VEL
LIN {X 0,Y 284.4,Z 343.682,A -85,B 0,C 180,E1 -16947.173,E2 -16947.173} C_VEL
LIN {X 0,Y 284.299,Z 343.696,A -85,B 0,C 180,E1 -16951.274,E2 -16951.274} C_VEL
LIN {X 0,Y 284.346,Z 343.693,A -85,B 0,C 180,E1 -16955.348,E2 -16955.348} C_VEL
LIN {X 0,Y 284.313,Z 343.686,A -85,B 0,C 180,E1 -16958.169,E2 -16958.169} C_VEL
LIN {X 0,Y 284.274,Z 343.698,A -85,B 0,C 180,E1 -16962.124,E2 -16962.124} C_VEL
LIN {X 0,Y 284.273,Z 343.696,A -85,B 0,C 180,E1 -16966.191,E2 -16966.191} C_VEL
LIN {X 0,Y 284.311,Z 343.694,A -85,B 0,C 180,E1 -16970.023,E2 -16970.023} C_VEL
LIN {X 0,Y 284.346,Z 343.805,A -85,B 0,C 180,E1 -16972.327,E2 -16972.327} C_VEL
LIN {X 0,Y 286.917,Z 354.647,A -85,B 0,C 180,E1 -16975.709,E2 -16975.709} C_VEL
LIN {X 0,Y 288.486,Z 361.682,A -85,B 0,C 180,E1 -16977.759,E2 -16977.759} C_VEL
LIN {X 0,Y 296.085,Z 381.417,A -85,B 0,C 180,E1 -16979.035,E2 -16979.035} C_VEL
LIN {X 0,Y 300.804,Z 412.872,A -85,B 0,C 180,E1 -16980.295,E2 -16980.295} C_VEL
LIN {X 0,Y 298.122,Z 499.987,A -85,B 0,C 180,E1 -16982.393,E2 -16982.393} C_VEL
LIN {X 0,Y 297.124,Z 514.638,A -85,B 0,C 180,E1 -16983.008,E2 -16983.008} C_VEL
LIN {X 0,Y 295.62,Z 529.222,A -85,B 0,C 180,E1 -16983.907,E2 -16983.907} C_VEL
LIN {X 0,Y 293.867,Z 543.056,A -85,B 0,C 180,E1 -16985.069,E2 -16985.069} C_VEL
LIN {X 0,Y 292.194,Z 555.504,A -85,B 0,C 180,E1 -16986.429,E2 -16986.429} C_VEL
LIN {X 0,Y 290.526,Z 565.685,A -85,B 0,C 180,E1 -16987.79,E2 -16987.79} C_VEL
LIN {X 0,Y 288.764,Z 575.341,A -85,B 0,C 180,E1 -16989.334,E2 -16989.334} C_VEL
LIN {X 0,Y 286.933,Z 586.098,A -85,B 0,C 180,E1 -16991.432,E2 -16991.432} C_VEL
LIN {X 0,Y 285.503,Z 594.948,A -85,B 0,C 180,E1 -16993.55,E2 -16993.55} C_VEL
LIN {X 0,Y 284.366,Z 602.314,A -85,B 0,C 180,E1 -16995.69,E2 -16995.69} C_VEL
LIN {X 0,Y 283.456,Z 608.407,A -85,B 0,C 180,E1 -16997.833,E2 -16997.833} C_VEL
LIN {X 0,Y 282.741,Z 614.883,A -85,B 0,C 180,E1 -17000.701,E2 -17000.701} C_VEL
LIN {X 0,Y 282.496,Z 618.598,A -85,B 0,C 180,E1 -17002.853,E2 -17002.853} C_VEL
LIN {X 0,Y 282.369,Z 622.208,A -85,B 0,C 180,E1 -17005.717,E2 -17005.717} C_VEL
LIN {X 0,Y 282.422,Z 623.47,A -85,B 0,C 180,E1 -17007.146,E2 -17007.146} C_VEL
LIN {X 0,Y 282.415,Z 624.944,A -85,B 0,C 180,E1 -17009.999,E2 -17009.999} C_VEL
LIN {X 0,Y 282.373,Z 625.058,A -85,B 0,C 180,E1 -17012.852,E2 -17012.852} C_VEL
LIN {X 0,Y 282.384,Z 623.837,A -85,B 0,C 180,E1 -17015.712,E2 -17015.712} C_VEL
LIN {X 0,Y 282.676,Z 621.278,A -85,B 0,C 180,E1 -17018.578,E2 -17018.578} C_VEL
LIN {X 0,Y 283.358,Z 617.314,A -85,B 0,C 180,E1 -17021.443,E2 -17021.443} C_VEL
LIN {X 0,Y 284.761,Z 611.814,A -85,B 0,C 180,E1 -17024.287,E2 -17024.287} C_VEL
LIN {X 0,Y 286.535,Z 604.643,A -85,B 0,C 180,E1 -17027.116,E2 -17027.116} C_VEL
LIN {X 0,Y 288.736,Z 596.776,A -85,B 0,C 180,E1 -17029.552,E2 -17029.552} C_VEL
LIN {X 0,Y 291.075,Z 588.594,A -85,B 0,C 180,E1 -17031.604,E2 -17031.604} C_VEL
LIN {X 0,Y 293.815,Z 578.777,A -85,B 0,C 180,E1 -17033.618,E2 -17033.618} C_VEL
LIN {X 0,Y 296.736,Z 567.578,A -85,B 0,C 180,E1 -17035.479,E2 -17035.479} C_VEL
LIN {X 0,Y 299.452,Z 555.908,A -85,B 0,C 180,E1 -17037.045,E2 -17037.045} C_VEL
LIN {X 0,Y 301.892,Z 544.099,A -85,B 0,C 180,E1 -17038.314,E2 -17038.314} C_VEL
LIN {X 0,Y 304.236,Z 531.168,A -85,B 0,C 180,E1 -17039.397,E2 -17039.397} C_VEL
LIN {X 0,Y 306.274,Z 517.159,A -85,B 0,C 180,E1 -17040.271,E2 -17040.271} C_VEL
LIN {X 0,Y 307.713,Z 503.492,A -85,B 0,C 180,E1 -17040.874,E2 -17040.874} C_VEL
LIN {X 0,Y 308.644,Z 486.815,A -85,B 0,C 180,E1 -17041.342,E2 -17041.342} C_VEL
LIN {X 0,Y 311.49,Z 415.393,A -85,B 0,C 180,E1 -17043.027,E2 -17043.027} C_VEL
LIN {X 0,Y 309.031,Z 400.123,A -85,B 0,C 180,E1 -17043.843,E2 -17043.843} C_VEL
LIN {X 0,Y 308.287,Z 396.895,A -85,B 0,C 180,E1 -17044.052,E2 -17044.052} C_VEL
LIN {X 0,Y 301.419,Z 382.17,A -85,B 0,C 180,E1 -17045.588,E2 -17045.588} C_VEL
LIN {X 0,Y 296.169,Z 372.308,A -85,B 0,C 180,E1 -17046.799,E2 -17046.799} C_VEL
LIN {X 0,Y 291.478,Z 363.988,A -85,B 0,C 180,E1 -17047.929,E2 -17047.929} C_VEL
LIN {X 0,Y 289.104,Z 359.546,A -85,B 0,C 180,E1 -17048.587,E2 -17048.587} C_VEL
LIN {X 0,Y 286.76,Z 351.501,A -85,B 0,C 180,E1 -17051.834,E2 -17051.834} C_VEL
LIN {X 0,Y 284.238,Z 343.688,A -85,B 0,C 180,E1 -17055.386,E2 -17055.386} C_VEL
LIN {X 0,Y 284.268,Z 343.703,A -85,B 0,C 180,E1 -17058.123,E2 -17058.123} C_VEL
LIN {X 0,Y 284.33,Z 343.689,A -85,B 0,C 180,E1 -17062.273,E2 -17062.273} C_VEL
LIN {X 0,Y 284.319,Z 343.695,A -85,B 0,C 180,E1 -17065.352,E2 -17065.352} C_VEL
LIN {X 0,Y 284.29,Z 343.698,A -85,B 0,C 180,E1 -17068.725,E2 -17068.725} C_VEL
LIN {X 0,Y 284.391,Z 343.68,A -85,B 0,C 180,E1 -17072.825,E2 -17072.825} C_VEL
LIN {X 0,Y 284.359,Z 343.68,A -85,B 0,C 180,E1 -17076.706,E2 -17076.706} C_VEL
LIN {X 0,Y 284.396,Z 343.674,A -85,B 0,C 180,E1 -17081.261,E2 -17081.261} C_VEL
LIN {X 0,Y 284.485,Z 343.663,A -85,B 0,C 180,E1 -17084.458,E2 -17084.458} C_VEL
LIN {X 0,Y 284.481,Z 343.662,A -85,B 0,C 180,E1 -17088.601,E2 -17088.601} C_VEL
LIN {X 0,Y 284.652,Z 343.653,A -85,B 0,C 180,E1 -17091.48,E2 -17091.48} C_VEL
LIN {X 0,Y 284.587,Z 343.657,A -85,B 0,C 180,E1 -17094.33,E2 -17094.33} C_VEL
LIN {X 0,Y 284.838,Z 343.628,A -85,B 0,C 180,E1 -17098.586,E2 -17098.586} C_VEL
LIN {X 0,Y 284.83,Z 343.62,A -85,B 0,C 180,E1 -17101.413,E2 -17101.413} C_VEL
LIN {X 0,Y 284.631,Z 343.655,A -85,B 0,C 180,E1 -17107.091,E2 -17107.091} C_VEL
LIN {X 0,Y 284.505,Z 343.666,A -85,B 0,C 180,E1 -17109.957,E2 -17109.957} C_VEL
LIN {X 0,Y 284.454,Z 343.678,A -85,B 0,C 180,E1 -17114.304,E2 -17114.304} C_VEL
LIN {X 0,Y 284.331,Z 343.688,A -85,B 0,C 180,E1 -17118.743,E2 -17118.743} C_VEL
LIN {X 0,Y 284.303,Z 343.691,A -85,B 0,C 180,E1 -17121.765,E2 -17121.765} C_VEL
LIN {X 0,Y 284.297,Z 343.693,A -85,B 0,C 180,E1 -17124.85,E2 -17124.85} C_VEL
LIN {X 0,Y 284.274,Z 343.683,A -85,B 0,C 180,E1 -17128.016,E2 -17128.016} C_VEL
LIN {X 0,Y 284.332,Z 343.686,A -85,B 0,C 180,E1 -17132.049,E2 -17132.049} C_VEL
LIN {X 0,Y 284.585,Z 344.941,A -85,B 0,C 180,E1 -17132.612,E2 -17132.612} C_VEL
LIN {X 0,Y 286.049,Z 347.541,A -85,B 0,C 180,E1 -17133.004,E2 -17133.004} C_VEL
LIN {X 0,Y 289.301,Z 352.108,A -85,B 0,C 180,E1 -17133.811,E2 -17133.811} C_VEL
LIN {X 0,Y 294.698,Z 360.47,A -85,B 0,C 180,E1 -17135.112,E2 -17135.112} C_VEL
LIN {X 0,Y 302.738,Z 374.319,A -85,B 0,C 180,E1 -17136.947,E2 -17136.947} C_VEL
LIN {X 0,Y 310.075,Z 388.911,A -85,B 0,C 180,E1 -17138.544,E2 -17138.544} C_VEL
LIN {X 0,Y 312.32,Z 393.801,A -85,B 0,C 180,E1 -17139.022,E2 -17139.022} C_VEL
LIN {X 0,Y 308.715,Z 479.783,A -85,B 0,C 180,E1 -17141.066,E2 -17141.066} C_VEL
LIN {X 0,Y 307.58,Z 494.169,A -85,B 0,C 180,E1 -17141.655,E2 -17141.655} C_VEL
LIN {X 0,Y 305.883,Z 507.828,A -85,B 0,C 180,E1 -17142.456,E2 -17142.456} C_VEL
LIN {X 0,Y 303.992,Z 520.817,A -85,B 0,C 180,E1 -17143.503,E2 -17143.503} C_VEL
LIN {X 0,Y 301.726,Z 532.913,A -85,B 0,C 180,E1 -17144.733,E2 -17144.733} C_VEL
LIN {X 0,Y 298.982,Z 545.416,A -85,B 0,C 180,E1 -17146.332,E2 -17146.332} C_VEL
LIN {X 0,Y 296.186,Z 556.71,A -85,B 0,C 180,E1 -17148.14,E2 -17148.14} C_VEL
LIN {X 0,Y 293.504,Z 566.785,A -85,B 0,C 180,E1 -17150.143,E2 -17150.143} C_VEL
LIN {X 0,Y 290.827,Z 575.939,A -85,B 0,C 180,E1 -17152.399,E2 -17152.399} C_VEL
LIN {X 0,Y 288.574,Z 583.354,A -85,B 0,C 180,E1 -17154.663,E2 -17154.663} C_VEL
LIN {X 0,Y 286.47,Z 590.265,A -85,B 0,C 180,E1 -17157.337,E2 -17157.337} C_VEL
LIN {X 0,Y 285.098,Z 594.913,A -85,B 0,C 180,E1 -17159.63,E2 -17159.63} C_VEL
LIN {X 0,Y 284.007,Z 598.565,A -85,B 0,C 180,E1 -17161.956,E2 -17161.956} C_VEL
LIN {X 0,Y 283.467,Z 600.423,A -85,B 0,C 180,E1 -17163.497,E2 -17163.497} C_VEL
LIN {X 0,Y 282.656,Z 602.919,A -85,B 0,C 180,E1 -17166.559,E2 -17166.559} C_VEL
LIN {X 0,Y 282.258,Z 603.906,A -85,B 0,C 180,E1 -17169.601,E2 -17169.601} C_VEL
LIN {X 0,Y 282.143,Z 603.439,A -85,B 0,C 180,E1 -17172.609,E2 -17172.609} C_VEL
LIN {X 0,Y 282.25,Z 601.549,A -85,B 0,C 180,E1 -17175.583,E2 -17175.583} C_VEL
LIN {X 0,Y 282.441,Z 600.061,A -85,B 0,C 180,E1 -17177.06,E2 -17177.06} C_VEL
LIN {X 0,Y 282.979,Z 595.934,A -85,B 0,C 180,E1 -17179.99,E2 -17179.99} C_VEL
LIN {X 0,Y 283.825,Z 590.215,A -85,B 0,C 180,E1 -17182.889,E2 -17182.889} C_VEL
LIN {X 0,Y 284.78,Z 583.782,A -85,B 0,C 180,E1 -17185.401,E2 -17185.401} C_VEL
LIN {X 0,Y 286.181,Z 575.77,A -85,B 0,C 180,E1 -17187.89,E2 -17187.89} C_VEL
LIN {X 0,Y 287.655,Z 567.395,A -85,B 0,C 180,E1 -17190.001,E2 -17190.001} C_VEL
LIN {X 0,Y 289.381,Z 557.32,A -85,B 0,C 180,E1 -17192.089,E2 -17192.089} C_VEL
LIN {X 0,Y 291.308,Z 546.046,A -85,B 0,C 180,E1 -17193.979,E2 -17193.979} C_VEL
LIN {X 0,Y 292.983,Z 534.852,A -85,B 0,C 180,E1 -17195.507,E2 -17195.507} C_VEL
LIN {X 0,Y 294.708,Z 522.613,A -85,B 0,C 180,E1 -17196.849,E2 -17196.849} C_VEL
LIN {X 0,Y 296.29,Z 509.05,A -85,B 0,C 180,E1 -17198.012,E2 -17198.012} C_VEL
LIN {X 0,Y 297.465,Z 494.945,A -85,B 0,C 180,E1 -17198.921,E2 -17198.921} C_VEL
LIN {X 0,Y 298.378,Z 481.019,A -85,B 0,C 180,E1 -17199.534,E2 -17199.534} C_VEL
LIN {X 0,Y 299.246,Z 457.321,A -85,B 0,C 180,E1 -17200.146,E2 -17200.146} C_VEL
LIN {X 0,Y 301.403,Z 384.567,A -85,B 0,C 180,E1 -17201.874,E2 -17201.874} C_VEL
LIN {X 0,Y 294.154,Z 365.547,A -85,B 0,C 180,E1 -17203.055,E2 -17203.055} C_VEL
LIN {X 0,Y 287.349,Z 350.102,A -85,B 0,C 180,E1 -17204.158,E2 -17204.158} C_VEL
LIN {X 0,Y 284.577,Z 344.387,A -85,B 0,C 180,E1 -17204.609,E2 -17204.609} C_VEL
LIN {X 0,Y 284.443,Z 343.681,A -85,B 0,C 180,E1 -17204.681,E2 -17204.681} C_VEL
LIN {X 0,Y 284.374,Z 343.692,A -85,B 0,C 180,E1 -17208.742,E2 -17208.742} C_VEL
LIN {X 0,Y 284.308,Z 343.697,A -85,B 0,C 180,E1 -17211.766,E2 -17211.766} C_VEL
LIN {X 0,Y 284.304,Z 343.698,A -85,B 0,C 180,E1 -17214.851,E2 -17214.851} C_VEL
LIN {X 0,Y 284.272,Z 343.698,A -85,B 0,C 180,E1 -17218.018,E2 -17218.018} C_VEL
LIN {X 0,Y 284.277,Z 343.699,A -85,B 0,C 180,E1 -17221.278,E2 -17221.278} C_VEL
LIN {X 0,Y 284.336,Z 343.686,A -85,B 0,C 180,E1 -17225.348,E2 -17225.348} C_VEL
LIN {X 0,Y 284.297,Z 343.691,A -85,B 0,C 180,E1 -17228.173,E2 -17228.173} C_VEL
LIN {X 0,Y 284.236,Z 343.701,A -85,B 0,C 180,E1 -17232.118,E2 -17232.118} C_VEL
LIN {X 0,Y 284.237,Z 343.695,A -85,B 0,C 180,E1 -17236.187,E2 -17236.187} C_VEL
LIN {X 0,Y 284.257,Z 343.699,A -85,B 0,C 180,E1 -17240.037,E2 -17240.037} C_VEL
LIN {X 0,Y 284.32,Z 343.676,A -85,B 0,C 180,E1 -17243.613,E2 -17243.613} C_VEL
LIN {X 0,Y 284.28,Z 343.694,A -85,B 0,C 180,E1 -17247.611,E2 -17247.611} C_VEL
LIN {X 0,Y 283.578,Z 343.787,A -85,B 0,C 180,E1 -17248.793,E2 -17248.793} C_VEL
LIN {X 0,Y 280.713,Z 344.141,A -85,B 0,C 180,E1 -17250.719,E2 -17250.719} C_VEL
LIN {X 0,Y 278.31,Z 344.439,A -85,B 0,C 180,E1 -17252.283,E2 -17252.283} C_VEL
LIN {X 0,Y 277.292,Z 344.565,A -85,B 0,C 180,E1 -17253.495,E2 -17253.495} C_VEL
LIN {X 0,Y 277.215,Z 344.576,A -85,B 0,C 180,E1 -17253.905,E2 -17253.905} C_VEL
LIN {X 0,Y 277.25,Z 344.57,A -85,B 0,C 180,E1 -17257.652,E2 -17257.652} C_VEL
LIN {X 0,Y 277.283,Z 344.569,A -85,B 0,C 180,E1 -17260.762,E2 -17260.762} C_VEL
LIN {X 0,Y 277.384,Z 344.546,A -85,B 0,C 180,E1 -17265.324,E2 -17265.324} C_VEL
LIN {X 0,Y 277.457,Z 344.536,A -85,B 0,C 180,E1 -17269.787,E2 -17269.787} C_VEL
LIN {X 0,Y 277.605,Z 344.528,A -85,B 0,C 180,E1 -17272.728,E2 -17272.728} C_VEL
LIN {X 0,Y 277.819,Z 344.485,A -85,B 0,C 180,E1 -17278.551,E2 -17278.551} C_VEL
LIN {X 0,Y 277.818,Z 344.49,A -85,B 0,C 180,E1 -17281.45,E2 -17281.45} C_VEL
LIN {X 0,Y 277.616,Z 344.526,A -85,B 0,C 180,E1 -17287.272,E2 -17287.272} C_VEL
LIN {X 0,Y 277.462,Z 344.548,A -85,B 0,C 180,E1 -17290.213,E2 -17290.213} C_VEL
LIN {X 0,Y 277.44,Z 344.547,A -85,B 0,C 180,E1 -17294.674,E2 -17294.674} C_VEL
LIN {X 0,Y 277.35,Z 344.559,A -85,B 0,C 180,E1 -17299.234,E2 -17299.234} C_VEL
LIN {X 0,Y 277.334,Z 344.56,A -85,B 0,C 180,E1 -17303.92,E2 -17303.92} C_VEL
LIN {X 0,Y 277.329,Z 344.566,A -85,B 0,C 180,E1 -17307.504,E2 -17307.504} C_VEL
LIN {X 0,Y 277.277,Z 344.567,A -85,B 0,C 180,E1 -17310.481,E2 -17310.481} C_VEL
LIN {X 0,Y 277.252,Z 344.573,A -85,B 0,C 180,E1 -17313.896,E2 -17313.896} C_VEL
LIN {X 0,Y 277.27,Z 344.565,A -85,B 0,C 180,E1 -17317.469,E2 -17317.469} C_VEL
LIN {X 0,Y 277.215,Z 344.581,A -85,B 0,C 180,E1 -17321.236,E2 -17321.236} C_VEL
LIN {X 0,Y 277.222,Z 344.58,A -85,B 0,C 180,E1 -17325.223,E2 -17325.223} C_VEL
LIN {X 0,Y 277.227,Z 344.576,A -85,B 0,C 180,E1 -17329.512,E2 -17329.512} C_VEL
LIN {X 0,Y 277.306,Z 344.776,A -85,B 0,C 180,E1 -17331.782,E2 -17331.782} C_VEL
LIN {X 0,Y 280.01,Z 356.01,A -85,B 0,C 180,E1 -17335.395,E2 -17335.395} C_VEL
LIN {X 0,Y 281.206,Z 361.31,A -85,B 0,C 180,E1 -17336.993,E2 -17336.993} C_VEL
LIN {X 0,Y 289.81,Z 383.316,A -85,B 0,C 180,E1 -17338.491,E2 -17338.491} C_VEL
LIN {X 0,Y 294.312,Z 414.085,A -85,B 0,C 180,E1 -17339.752,E2 -17339.752} C_VEL
LIN {X 0,Y 291.584,Z 499.981,A -85,B 0,C 180,E1 -17341.866,E2 -17341.866} C_VEL
LIN {X 0,Y 290.534,Z 514.544,A -85,B 0,C 180,E1 -17342.491,E2 -17342.491} C_VEL
LIN {X 0,Y 289.065,Z 528.524,A -85,B 0,C 180,E1 -17343.366,E2 -17343.366} C_VEL
LIN {X 0,Y 287.295,Z 542.094,A -85,B 0,C 180,E1 -17344.516,E2 -17344.516} C_VEL
LIN {X 0,Y 285.608,Z 554.316,A -85,B 0,C 180,E1 -17345.859,E2 -17345.859} C_VEL
LIN {X 0,Y 283.88,Z 564.612,A -85,B 0,C 180,E1 -17347.242,E2 -17347.242} C_VEL
LIN {X 0,Y 282.043,Z 574.409,A -85,B 0,C 180,E1 -17348.818,E2 -17348.818} C_VEL
LIN {X 0,Y 280.125,Z 585.279,A -85,B 0,C 180,E1 -17350.963,E2 -17350.963} C_VEL
LIN {X 0,Y 278.624,Z 594.242,A -85,B 0,C 180,E1 -17353.137,E2 -17353.137} C_VEL
LIN {X 0,Y 277.454,Z 601.672,A -85,B 0,C 180,E1 -17355.326,E2 -17355.326} C_VEL
LIN {X 0,Y 276.468,Z 607.835,A -85,B 0,C 180,E1 -17357.52,E2 -17357.52} C_VEL
LIN {X 0,Y 275.673,Z 614.374,A -85,B 0,C 180,E1 -17360.46,E2 -17360.46} C_VEL
LIN {X 0,Y 275.365,Z 619.23,A -85,B 0,C 180,E1 -17363.404,E2 -17363.404} C_VEL
LIN {X 0,Y 275.279,Z 621.818,A -85,B 0,C 180,E1 -17365.606,E2 -17365.606} C_VEL
LIN {X 0,Y 275.326,Z 623.108,A -85,B 0,C 180,E1 -17367.072,E2 -17367.072} C_VEL
LIN {X 0,Y 275.334,Z 624.636,A -85,B 0,C 180,E1 -17369.999,E2 -17369.999} C_VEL
LIN {X 0,Y 275.279,Z 624.801,A -85,B 0,C 180,E1 -17372.926,E2 -17372.926} C_VEL
LIN {X 0,Y 275.296,Z 623.63,A -85,B 0,C 180,E1 -17375.86,E2 -17375.86} C_VEL
LIN {X 0,Y 275.625,Z 621.127,A -85,B 0,C 180,E1 -17378.799,E2 -17378.799} C_VEL
LIN {X 0,Y 276.352,Z 617.237,A -85,B 0,C 180,E1 -17381.737,E2 -17381.737} C_VEL
LIN {X 0,Y 277.839,Z 611.825,A -85,B 0,C 180,E1 -17384.651,E2 -17384.651} C_VEL
LIN {X 0,Y 279.738,Z 604.723,A -85,B 0,C 180,E1 -17387.545,E2 -17387.545} C_VEL
LIN {X 0,Y 282.032,Z 596.935,A -85,B 0,C 180,E1 -17390.036,E2 -17390.036} C_VEL
LIN {X 0,Y 284.499,Z 588.84,A -85,B 0,C 180,E1 -17392.129,E2 -17392.129} C_VEL
LIN {X 0,Y 287.328,Z 579.126,A -85,B 0,C 180,E1 -17394.185,E2 -17394.185} C_VEL
LIN {X 0,Y 290.344,Z 568.113,A -85,B 0,C 180,E1 -17396.072,E2 -17396.072} C_VEL
LIN {X 0,Y 293.182,Z 556.558,A -85,B 0,C 180,E1 -17397.673,E2 -17397.673} C_VEL
LIN {X 0,Y 295.715,Z 544.971,A -85,B 0,C 180,E1 -17398.961,E2 -17398.961} C_VEL
LIN {X 0,Y 297.738,Z 534.349,A -85,B 0,C 180,E1 -17399.909,E2 -17399.909} C_VEL
LIN {X 0,Y 299.968,Z 520.916,A -85,B 0,C 180,E1 -17400.83,E2 -17400.83} C_VEL
LIN {X 0,Y 301.547,Z 508.05,A -85,B 0,C 180,E1 -17401.479,E2 -17401.479} C_VEL
LIN {X 0,Y 302.593,Z 494.588,A -85,B 0,C 180,E1 -17401.944,E2 -17401.944} C_VEL
LIN {X 0,Y 305.877,Z 416.364,A -85,B 0,C 180,E1 -17403.827,E2 -17403.827} C_VEL
LIN {X 0,Y 303.399,Z 400.976,A -85,B 0,C 180,E1 -17404.681,E2 -17404.681} C_VEL
LIN {X 0,Y 298.076,Z 388.976,A -85,B 0,C 180,E1 -17405.929,E2 -17405.929} C_VEL
LIN {X 0,Y 292.584,Z 378.243,A -85,B 0,C 180,E1 -17407.24,E2 -17407.24} C_VEL
LIN {X 0,Y 287.097,Z 368.477,A -85,B 0,C 180,E1 -17408.61,E2 -17408.61} C_VEL
LIN {X 0,Y 284.118,Z 363.438,A -85,B 0,C 180,E1 -17409.38,E2 -17409.38} C_VEL
LIN {X 0,Y 281.795,Z 359.268,A -85,B 0,C 180,E1 -17410.022,E2 -17410.022} C_VEL
LIN {X 0,Y 279.563,Z 351.904,A -85,B 0,C 180,E1 -17413.194,E2 -17413.194} C_VEL
LIN {X 0,Y 277.184,Z 344.568,A -85,B 0,C 180,E1 -17416.706,E2 -17416.706} C_VEL
LIN {X 0,Y 277.233,Z 344.553,A -85,B 0,C 180,E1 -17420.671,E2 -17420.671} C_VEL
LIN {X 0,Y 277.298,Z 344.563,A -85,B 0,C 180,E1 -17424.343,E2 -17424.343} C_VEL
LIN {X 0,Y 277.239,Z 344.571,A -85,B 0,C 180,E1 -17427.835,E2 -17427.835} C_VEL
LIN {X 0,Y 277.284,Z 344.567,A -85,B 0,C 180,E1 -17431.211,E2 -17431.211} C_VEL
LIN {X 0,Y 277.307,Z 344.562,A -85,B 0,C 180,E1 -17434.478,E2 -17434.478} C_VEL
LIN {X 0,Y 277.278,Z 344.561,A -85,B 0,C 180,E1 -17437.654,E2 -17437.654} C_VEL
LIN {X 0,Y 277.338,Z 344.553,A -85,B 0,C 180,E1 -17440.765,E2 -17440.765} C_VEL
LIN {X 0,Y 277.428,Z 344.541,A -85,B 0,C 180,E1 -17445.325,E2 -17445.325} C_VEL
LIN {X 0,Y 277.499,Z 344.534,A -85,B 0,C 180,E1 -17449.788,E2 -17449.788} C_VEL
LIN {X 0,Y 277.645,Z 344.514,A -85,B 0,C 180,E1 -17452.728,E2 -17452.728} C_VEL
LIN {X 0,Y 277.804,Z 344.504,A -85,B 0,C 180,E1 -17458.55,E2 -17458.55} C_VEL
LIN {X 0,Y 277.797,Z 344.496,A -85,B 0,C 180,E1 -17461.449,E2 -17461.449} C_VEL
LIN {X 0,Y 277.59,Z 344.534,A -85,B 0,C 180,E1 -17467.272,E2 -17467.272} C_VEL
LIN {X 0,Y 277.448,Z 344.547,A -85,B 0,C 180,E1 -17470.213,E2 -17470.213} C_VEL
LIN {X 0,Y 277.4,Z 344.557,A -85,B 0,C 180,E1 -17474.675,E2 -17474.675} C_VEL
LIN {X 0,Y 277.295,Z 344.563,A -85,B 0,C 180,E1 -17479.237,E2 -17479.237} C_VEL
LIN {X 0,Y 277.273,Z 344.573,A -85,B 0,C 180,E1 -17483.925,E2 -17483.925} C_VEL
LIN {X 0,Y 277.261,Z 344.561,A -85,B 0,C 180,E1 -17487.483,E2 -17487.483} C_VEL
LIN {X 0,Y 277.23,Z 344.617,A -85,B 0,C 180,E1 -17490.77,E2 -17490.77} C_VEL
LIN {X 0,Y 277.384,Z 345.397,A -85,B 0,C 180,E1 -17491.079,E2 -17491.079} C_VEL
LIN {X 0,Y 278.625,Z 347.992,A -85,B 0,C 180,E1 -17491.453,E2 -17491.453} C_VEL
LIN {X 0,Y 280.697,Z 350.244,A -85,B 0,C 180,E1 -17491.989,E2 -17491.989} C_VEL
LIN {X 0,Y 283.185,Z 353.97,A -85,B 0,C 180,E1 -17492.651,E2 -17492.651} C_VEL
LIN {X 0,Y 288.43,Z 362.008,A -85,B 0,C 180,E1 -17493.989,E2 -17493.989} C_VEL
LIN {X 0,Y 294.304,Z 371.68,A -85,B 0,C 180,E1 -17495.414,E2 -17495.414} C_VEL
LIN {X 0,Y 301.609,Z 385.324,A -85,B 0,C 180,E1 -17497.108,E2 -17497.108} C_VEL
LIN {X 0,Y 306.71,Z 396.114,A -85,B 0,C 180,E1 -17498.251,E2 -17498.251} C_VEL
LIN {X 0,Y 302.973,Z 480.988,A -85,B 0,C 180,E1 -17500.307,E2 -17500.307} C_VEL
LIN {X 0,Y 301.74,Z 495.293,A -85,B 0,C 180,E1 -17500.913,E2 -17500.913} C_VEL
LIN {X 0,Y 299.875,Z 509.65,A -85,B 0,C 180,E1 -17501.794,E2 -17501.794} C_VEL
LIN {X 0,Y 298.044,Z 521.529,A -85,B 0,C 180,E1 -17502.785,E2 -17502.785} C_VEL
LIN {X 0,Y 295.554,Z 534.111,A -85,B 0,C 180,E1 -17504.099,E2 -17504.099} C_VEL
LIN {X 0,Y 292.829,Z 545.945,A -85,B 0,C 180,E1 -17505.655,E2 -17505.655} C_VEL
LIN {X 0,Y 289.899,Z 557.17,A -85,B 0,C 180,E1 -17507.488,E2 -17507.488} C_VEL
LIN {X 0,Y 287.37,Z 566.159,A -85,B 0,C 180,E1 -17509.3,E2 -17509.3} C_VEL
LIN {X 0,Y 284.702,Z 574.943,A -85,B 0,C 180,E1 -17511.444,E2 -17511.444} C_VEL
LIN {X 0,Y 282.289,Z 582.598,A -85,B 0,C 180,E1 -17513.753,E2 -17513.753} C_VEL
LIN {X 0,Y 279.994,Z 589.754,A -85,B 0,C 180,E1 -17516.483,E2 -17516.483} C_VEL
LIN {X 0,Y 278.234,Z 595.183,A -85,B 0,C 180,E1 -17519.183,E2 -17519.183} C_VEL
LIN {X 0,Y 277.209,Z 598.327,A -85,B 0,C 180,E1 -17521.205,E2 -17521.205} C_VEL
LIN {X 0,Y 276.633,Z 600.3,A -85,B 0,C 180,E1 -17522.789,E2 -17522.789} C_VEL
LIN {X 0,Y 276.081,Z 601.859,A -85,B 0,C 180,E1 -17524.359,E2 -17524.359} C_VEL
LIN {X 0,Y 275.543,Z 603.386,A -85,B 0,C 180,E1 -17526.665,E2 -17526.665} C_VEL
LIN {X 0,Y 275.217,Z 604.146,A -85,B 0,C 180,E1 -17529.054,E2 -17529.054} C_VEL
LIN {X 0,Y 275.05,Z 603.832,A -85,B 0,C 180,E1 -17532.146,E2 -17532.146} C_VEL
LIN {X 0,Y 275.105,Z 602.094,A -85,B 0,C 180,E1 -17535.2,E2 -17535.2} C_VEL
LIN {X 0,Y 275.324,Z 600.683,A -85,B 0,C 180,E1 -17536.72,E2 -17536.72} C_VEL
LIN {X 0,Y 275.811,Z 596.775,A -85,B 0,C 180,E1 -17539.727,E2 -17539.727} C_VEL
LIN {X 0,Y 276.556,Z 592.024,A -85,B 0,C 180,E1 -17542.341,E2 -17542.341} C_VEL
LIN {X 0,Y 277.633,Z 584.99,A -85,B 0,C 180,E1 -17545.282,E2 -17545.282} C_VEL
LIN {X 0,Y 279.032,Z 577.179,A -85,B 0,C 180,E1 -17547.836,E2 -17547.836} C_VEL
LIN {X 0,Y 280.504,Z 569.036,A -85,B 0,C 180,E1 -17550.001,E2 -17550.001} C_VEL
LIN {X 0,Y 282.255,Z 559.222,A -85,B 0,C 180,E1 -17552.142,E2 -17552.142} C_VEL
LIN {X 0,Y 284.209,Z 548.303,A -85,B 0,C 180,E1 -17554.078,E2 -17554.078} C_VEL
LIN {X 0,Y 286.121,Z 536.222,A -85,B 0,C 180,E1 -17555.817,E2 -17555.817} C_VEL
LIN {X 0,Y 287.866,Z 524.277,A -85,B 0,C 180,E1 -17557.189,E2 -17557.189} C_VEL
LIN {X 0,Y 289.488,Z 511.142,A -85,B 0,C 180,E1 -17558.377,E2 -17558.377} C_VEL
LIN {X 0,Y 290.815,Z 496.85,A -85,B 0,C 180,E1 -17559.346,E2 -17559.346} C_VEL
LIN {X 0,Y 291.778,Z 482.637,A -85,B 0,C 180,E1 -17560.014,E2 -17560.014} C_VEL
LIN {X 0,Y 292.534,Z 463.194,A -85,B 0,C 180,E1 -17560.557,E2 -17560.557} C_VEL
LIN {X 0,Y 295.035,Z 386.32,A -85,B 0,C 180,E1 -17562.407,E2 -17562.407} C_VEL
LIN {X 0,Y 287.481,Z 366.74,A -85,B 0,C 180,E1 -17563.678,E2 -17563.678} C_VEL
LIN {X 0,Y 281.407,Z 353.181,A -85,B 0,C 180,E1 -17564.694,E2 -17564.694} C_VEL
LIN {X 0,Y 277.637,Z 345.648,A -85,B 0,C 180,E1 -17565.325,E2 -17565.325} C_VEL
LIN {X 0,Y 277.412,Z 344.559,A -85,B 0,C 180,E1 -17565.382,E2 -17565.382} C_VEL
LIN {X 0,Y 277.323,Z 344.572,A -85,B 0,C 180,E1 -17569.237,E2 -17569.237} C_VEL
LIN {X 0,Y 277.281,Z 344.571,A -85,B 0,C 180,E1 -17573.926,E2 -17573.926} C_VEL
LIN {X 0,Y 277.265,Z 344.573,A -85,B 0,C 180,E1 -17577.482,E2 -17577.482} C_VEL
LIN {X 0,Y 277.237,Z 344.574,A -85,B 0,C 180,E1 -17582.166,E2 -17582.166} C_VEL
LIN {X 0,Y 277.273,Z 344.564,A -85,B 0,C 180,E1 -17585.798,E2 -17585.798} C_VEL
LIN {X 0,Y 277.216,Z 344.578,A -85,B 0,C 180,E1 -17589.332,E2 -17589.332} C_VEL
LIN {X 0,Y 277.191,Z 344.571,A -85,B 0,C 180,E1 -17593.203,E2 -17593.203} C_VEL
LIN {X 0,Y 277.192,Z 344.578,A -85,B 0,C 180,E1 -17597.332,E2 -17597.332} C_VEL
LIN {X 0,Y 277.224,Z 344.569,A -85,B 0,C 180,E1 -17601.805,E2 -17601.805} C_VEL
LIN {X 0,Y 277.278,Z 344.553,A -85,B 0,C 180,E1 -17604.341,E2 -17604.341} C_VEL
LIN {X 0,Y 277.239,Z 344.572,A -85,B 0,C 180,E1 -17607.836,E2 -17607.836} C_VEL
LIN {X 0,Y 277.218,Z 344.574,A -85,B 0,C 180,E1 -17611.205,E2 -17611.205} C_VEL
LIN {X 0,Y 277.215,Z 344.576,A -85,B 0,C 180,E1 -17613.905,E2 -17613.905} C_VEL
LIN {X 0,Y 276.575,Z 344.661,A -85,B 0,C 180,E1 -17615.117,E2 -17615.117} C_VEL
LIN {X 0,Y 273.778,Z 345.016,A -85,B 0,C 180,E1 -17617.093,E2 -17617.093} C_VEL
LIN {X 0,Y 271.375,Z 345.313,A -85,B 0,C 180,E1 -17618.697,E2 -17618.697} C_VEL
LIN {X 0,Y 270.317,Z 345.439,A -85,B 0,C 180,E1 -17619.94,E2 -17619.94} C_VEL
LIN {X 0,Y 270.217,Z 345.449,A -85,B 0,C 180,E1 -17620.361,E2 -17620.361} C_VEL
LIN {X 0,Y 270.347,Z 345.423,A -85,B 0,C 180,E1 -17624.933,E2 -17624.933} C_VEL
LIN {X 0,Y 270.389,Z 345.414,A -85,B 0,C 180,E1 -17629.517,E2 -17629.517} C_VEL
LIN {X 0,Y 270.567,Z 345.406,A -85,B 0,C 180,E1 -17632.538,E2 -17632.538} C_VEL
LIN {X 0,Y 270.784,Z 345.36,A -85,B 0,C 180,E1 -17638.513,E2 -17638.513} C_VEL
LIN {X 0,Y 270.782,Z 345.365,A -85,B 0,C 180,E1 -17641.488,E2 -17641.488} C_VEL
LIN {X 0,Y 270.576,Z 345.404,A -85,B 0,C 180,E1 -17647.463,E2 -17647.463} C_VEL
LIN {X 0,Y 270.415,Z 345.424,A -85,B 0,C 180,E1 -17650.483,E2 -17650.483} C_VEL
LIN {X 0,Y 270.408,Z 345.423,A -85,B 0,C 180,E1 -17655.065,E2 -17655.065} C_VEL
LIN {X 0,Y 270.307,Z 345.435,A -85,B 0,C 180,E1 -17659.756,E2 -17659.756} C_VEL
LIN {X 0,Y 270.279,Z 345.436,A -85,B 0,C 180,E1 -17664.586,E2 -17664.586} C_VEL
LIN {X 0,Y 270.275,Z 345.441,A -85,B 0,C 180,E1 -17667.909,E2 -17667.909} C_VEL
LIN {X 0,Y 270.189,Z 345.454,A -85,B 0,C 180,E1 -17671.348,E2 -17671.348} C_VEL
LIN {X 0,Y 270.207,Z 345.451,A -85,B 0,C 180,E1 -17674.905,E2 -17674.905} C_VEL
LIN {X 0,Y 270.203,Z 345.444,A -85,B 0,C 180,E1 -17678.71,E2 -17678.71} C_VEL
LIN {X 0,Y 270.177,Z 345.458,A -85,B 0,C 180,E1 -17683.25,E2 -17683.25} C_VEL
LIN {X 0,Y 270.18,Z 345.453,A -85,B 0,C 180,E1 -17687.442,E2 -17687.442} C_VEL
LIN {X 0,Y 270.25,Z 345.595,A -85,B 0,C 180,E1 -17691.166,E2 -17691.166} C_VEL
LIN {X 0,Y 272.743,Z 355.813,A -85,B 0,C 180,E1 -17694.565,E2 -17694.565} C_VEL
LIN {X 0,Y 273.889,Z 360.858,A -85,B 0,C 180,E1 -17696.174,E2 -17696.174} C_VEL
LIN {X 0,Y 282.545,Z 382.776,A -85,B 0,C 180,E1 -17697.749,E2 -17697.749} C_VEL
LIN {X 0,Y 283.85,Z 386.811,A -85,B 0,C 180,E1 -17697.997,E2 -17697.997} C_VEL
LIN {X 0,Y 287.876,Z 414.111,A -85,B 0,C 180,E1 -17699.156,E2 -17699.156} C_VEL
LIN {X 0,Y 285.065,Z 499.875,A -85,B 0,C 180,E1 -17701.314,E2 -17701.314} C_VEL
LIN {X 0,Y 283.985,Z 514.386,A -85,B 0,C 180,E1 -17701.951,E2 -17701.951} C_VEL
LIN {X 0,Y 282.401,Z 528.906,A -85,B 0,C 180,E1 -17702.886,E2 -17702.886} C_VEL
LIN {X 0,Y 280.645,Z 541.797,A -85,B 0,C 180,E1 -17704.007,E2 -17704.007} C_VEL
LIN {X 0,Y 279.026,Z 553.43,A -85,B 0,C 180,E1 -17705.308,E2 -17705.308} C_VEL
LIN {X 0,Y 277.243,Z 563.488,A -85,B 0,C 180,E1 -17706.665,E2 -17706.665} C_VEL
LIN {X 0,Y 275.006,Z 575.419,A -85,B 0,C 180,E1 -17708.642,E2 -17708.642} C_VEL
LIN {X 0,Y 273.06,Z 586.082,A -85,B 0,C 180,E1 -17710.842,E2 -17710.842} C_VEL
LIN {X 0,Y 271.503,Z 594.864,A -85,B 0,C 180,E1 -17713.068,E2 -17713.068} C_VEL
LIN {X 0,Y 270.093,Z 603.245,A -85,B 0,C 180,E1 -17715.687,E2 -17715.687} C_VEL
LIN {X 0,Y 269.169,Z 609.088,A -85,B 0,C 180,E1 -17717.942,E2 -17717.942} C_VEL
LIN {X 0,Y 268.618,Z 613.859,A -85,B 0,C 180,E1 -17720.207,E2 -17720.207} C_VEL
LIN {X 0,Y 268.351,Z 617.7,A -85,B 0,C 180,E1 -17722.474,E2 -17722.474} C_VEL
LIN {X 0,Y 268.194,Z 621.426,A -85,B 0,C 180,E1 -17725.49,E2 -17725.49} C_VEL
LIN {X 0,Y 268.233,Z 622.743,A -85,B 0,C 180,E1 -17726.995,E2 -17726.995} C_VEL
LIN {X 0,Y 268.255,Z 624.326,A -85,B 0,C 180,E1 -17729.999,E2 -17729.999} C_VEL
LIN {X 0,Y 268.188,Z 624.544,A -85,B 0,C 180,E1 -17733.003,E2 -17733.003} C_VEL
LIN {X 0,Y 268.219,Z 623.429,A -85,B 0,C 180,E1 -17736.015,E2 -17736.015} C_VEL
LIN {X 0,Y 268.559,Z 620.982,A -85,B 0,C 180,E1 -17739.032,E2 -17739.032} C_VEL
LIN {X 0,Y 269.354,Z 617.152,A -85,B 0,C 180,E1 -17742.047,E2 -17742.047} C_VEL
LIN {X 0,Y 270.914,Z 611.832,A -85,B 0,C 180,E1 -17745.034,E2 -17745.034} C_VEL
LIN {X 0,Y 272.382,Z 606.592,A -85,B 0,C 180,E1 -17747.315,E2 -17747.315} C_VEL
LIN {X 0,Y 274.597,Z 599.476,A -85,B 0,C 180,E1 -17749.822,E2 -17749.822} C_VEL
LIN {X 0,Y 276.983,Z 591.931,A -85,B 0,C 180,E1 -17751.977,E2 -17751.977} C_VEL
LIN {X 0,Y 279.863,Z 582.912,A -85,B 0,C 180,E1 -17754.082,E2 -17754.082} C_VEL
LIN {X 0,Y 283.065,Z 572.039,A -85,B 0,C 180,E1 -17756.147,E2 -17756.147} C_VEL
LIN {X 0,Y 285.953,Z 561.047,A -85,B 0,C 180,E1 -17757.836,E2 -17757.836} C_VEL
LIN {X 0,Y 288.936,Z 548.989,A -85,B 0,C 180,E1 -17759.307,E2 -17759.307} C_VEL
LIN {X 0,Y 291.27,Z 537.464,A -85,B 0,C 180,E1 -17760.443,E2 -17760.443} C_VEL
LIN {X 0,Y 293.766,Z 523.844,A -85,B 0,C 180,E1 -17761.454,E2 -17761.454} C_VEL
LIN {X 0,Y 295.676,Z 509.573,A -85,B 0,C 180,E1 -17762.228,E2 -17762.228} C_VEL
LIN {X 0,Y 296.901,Z 495.755,A -85,B 0,C 180,E1 -17762.732,E2 -17762.732} C_VEL
LIN {X 0,Y 300.347,Z 417.704,A -85,B 0,C 180,E1 -17764.642,E2 -17764.642} C_VEL
LIN {X 0,Y 298.204,Z 403.802,A -85,B 0,C 180,E1 -17765.432,E2 -17765.432} C_VEL
LIN {X 0,Y 292.038,Z 390.308,A -85,B 0,C 180,E1 -17766.936,E2 -17766.936} C_VEL
LIN {X 0,Y 286.015,Z 378.628,A -85,B 0,C 180,E1 -17768.462,E2 -17768.462} C_VEL
LIN {X 0,Y 280.071,Z 368.338,A -85,B 0,C 180,E1 -17770.038,E2 -17770.038} C_VEL
LIN {X 0,Y 277.205,Z 363.602,A -85,B 0,C 180,E1 -17770.832,E2 -17770.832} C_VEL
LIN {X 0,Y 274.43,Z 358.908,A -85,B 0,C 180,E1 -17771.635,E2 -17771.635} C_VEL
LIN {X 0,Y 271.679,Z 350.176,A -85,B 0,C 180,E1 -17775.696,E2 -17775.696} C_VEL
LIN {X 0,Y 270.159,Z 345.459,A -85,B 0,C 180,E1 -17778.168,E2 -17778.168} C_VEL
LIN {X 0,Y 270.202,Z 345.433,A -85,B 0,C 180,E1 -17781.373,E2 -17781.373} C_VEL
LIN {X 0,Y 270.21,Z 345.449,A -85,B 0,C 180,E1 -17785.095,E2 -17785.095} C_VEL
LIN {X 0,Y 270.195,Z 345.452,A -85,B 0,C 180,E1 -17789.129,E2 -17789.129} C_VEL
LIN {X 0,Y 270.259,Z 345.446,A -85,B 0,C 180,E1 -17792.144,E2 -17792.144} C_VEL
LIN {X 0,Y 270.271,Z 345.445,A -85,B 0,C 180,E1 -17795.518,E2 -17795.518} C_VEL
LIN {X 0,Y 270.295,Z 345.433,A -85,B 0,C 180,E1 -17800.243,E2 -17800.243} C_VEL
LIN {X 0,Y 270.396,Z 345.416,A -85,B 0,C 180,E1 -17804.934,E2 -17804.934} C_VEL
LIN {X 0,Y 270.434,Z 345.412,A -85,B 0,C 180,E1 -17809.518,E2 -17809.518} C_VEL
LIN {X 0,Y 270.603,Z 345.392,A -85,B 0,C 180,E1 -17812.538,E2 -17812.538} C_VEL
LIN {X 0,Y 270.769,Z 345.379,A -85,B 0,C 180,E1 -17818.512,E2 -17818.512} C_VEL
LIN {X 0,Y 270.763,Z 345.372,A -85,B 0,C 180,E1 -17821.487,E2 -17821.487} C_VEL
LIN {X 0,Y 270.552,Z 345.41,A -85,B 0,C 180,E1 -17827.462,E2 -17827.462} C_VEL
LIN {X 0,Y 270.401,Z 345.428,A -85,B 0,C 180,E1 -17830.482,E2 -17830.482} C_VEL
LIN {X 0,Y 270.359,Z 345.431,A -85,B 0,C 180,E1 -17835.067,E2 -17835.067} C_VEL
LIN {X 0,Y 270.243,Z 345.442,A -85,B 0,C 180,E1 -17839.759,E2 -17839.759} C_VEL
LIN {X 0,Y 270.215,Z 345.448,A -85,B 0,C 180,E1 -17844.591,E2 -17844.591} C_VEL
LIN {X 0,Y 270.199,Z 345.434,A -85,B 0,C 180,E1 -17848.763,E2 -17848.763} C_VEL
LIN {X 0,Y 270.185,Z 345.548,A -85,B 0,C 180,E1 -17849.35,E2 -17849.35} C_VEL
LIN {X 0,Y 271.257,Z 348.427,A -85,B 0,C 180,E1 -17849.765,E2 -17849.765} C_VEL
LIN {X 0,Y 273.683,Z 351.016,A -85,B 0,C 180,E1 -17850.449,E2 -17850.449} C_VEL
LIN {X 0,Y 275.807,Z 354.324,A -85,B 0,C 180,E1 -17851.064,E2 -17851.064} C_VEL
LIN {X 0,Y 277.15,Z 355.963,A -85,B 0,C 180,E1 -17851.427,E2 -17851.427} C_VEL
LIN {X 0,Y 283.299,Z 365.118,A -85,B 0,C 180,E1 -17853.077,E2 -17853.077} C_VEL
LIN {X 0,Y 290.141,Z 376.612,A -85,B 0,C 180,E1 -17854.821,E2 -17854.821} C_VEL
LIN {X 0,Y 297.177,Z 389.966,A -85,B 0,C 180,E1 -17856.515,E2 -17856.515} C_VEL
LIN {X 0,Y 301.166,Z 398.475,A -85,B 0,C 180,E1 -17857.451,E2 -17857.451} C_VEL
LIN {X 0,Y 297.362,Z 481.072,A -85,B 0,C 180,E1 -17859.478,E2 -17859.478} C_VEL
LIN {X 0,Y 296.161,Z 494.876,A -85,B 0,C 180,E1 -17860.064,E2 -17860.064} C_VEL
LIN {X 0,Y 294.412,Z 508.038,A -85,B 0,C 180,E1 -17860.853,E2 -17860.853} C_VEL
LIN {X 0,Y 292.275,Z 521.446,A -85,B 0,C 180,E1 -17861.959,E2 -17861.959} C_VEL
LIN {X 0,Y 289.682,Z 534.138,A -85,B 0,C 180,E1 -17863.297,E2 -17863.297} C_VEL
LIN {X 0,Y 287.038,Z 545.238,A -85,B 0,C 180,E1 -17864.763,E2 -17864.763} C_VEL
LIN {X 0,Y 283.954,Z 556.626,A -85,B 0,C 180,E1 -17866.623,E2 -17866.623} C_VEL
LIN {X 0,Y 281.109,Z 566.332,A -85,B 0,C 180,E1 -17868.592,E2 -17868.592} C_VEL
LIN {X 0,Y 278.235,Z 575.365,A -85,B 0,C 180,E1 -17870.843,E2 -17870.843} C_VEL
LIN {X 0,Y 275.666,Z 582.98,A -85,B 0,C 180,E1 -17873.195,E2 -17873.195} C_VEL
LIN {X 0,Y 273.564,Z 589.181,A -85,B 0,C 180,E1 -17875.586,E2 -17875.586} C_VEL
LIN {X 0,Y 271.856,Z 594.174,A -85,B 0,C 180,E1 -17878,E2 -17878} C_VEL
LIN {X 0,Y 270.494,Z 598.089,A -85,B 0,C 180,E1 -17880.42,E2 -17880.42} C_VEL
LIN {X 0,Y 269.696,Z 600.53,A -85,B 0,C 180,E1 -17882.374,E2 -17882.374} C_VEL
LIN {X 0,Y 268.75,Z 603.04,A -85,B 0,C 180,E1 -17885.267,E2 -17885.267} C_VEL
LIN {X 0,Y 268.171,Z 604.387,A -85,B 0,C 180,E1 -17888.477,E2 -17888.477} C_VEL
LIN {X 0,Y 267.961,Z 604.224,A -85,B 0,C 180,E1 -17891.657,E2 -17891.657} C_VEL
LIN {X 0,Y 267.987,Z 602.632,A -85,B 0,C 180,E1 -17894.798,E2 -17894.798} C_VEL
LIN {X 0,Y 268.194,Z 601.295,A -85,B 0,C 180,E1 -17896.36,E2 -17896.36} C_VEL
LIN {X 0,Y 268.673,Z 597.538,A -85,B 0,C 180,E1 -17899.451,E2 -17899.451} C_VEL
LIN {X 0,Y 269.498,Z 592.235,A -85,B 0,C 180,E1 -17902.509,E2 -17902.509} C_VEL
LIN {X 0,Y 270.315,Z 587.094,A -85,B 0,C 180,E1 -17904.78,E2 -17904.78} C_VEL
LIN {X 0,Y 271.617,Z 579.757,A -85,B 0,C 180,E1 -17907.406,E2 -17907.406} C_VEL
LIN {X 0,Y 273.374,Z 570.647,A -85,B 0,C 180,E1 -17910.001,E2 -17910.001} C_VEL
LIN {X 0,Y 275.146,Z 561.097,A -85,B 0,C 180,E1 -17912.197,E2 -17912.197} C_VEL
LIN {X 0,Y 277.021,Z 550.528,A -85,B 0,C 180,E1 -17914.184,E2 -17914.184} C_VEL
LIN {X 0,Y 279.029,Z 538.825,A -85,B 0,C 180,E1 -17915.965,E2 -17915.965} C_VEL
LIN {X 0,Y 280.816,Z 527.395,A -85,B 0,C 180,E1 -17917.371,E2 -17917.371} C_VEL
LIN {X 0,Y 282.468,Z 515.041,A -85,B 0,C 180,E1 -17918.587,E2 -17918.587} C_VEL
LIN {X 0,Y 283.889,Z 501.425,A -85,B 0,C 180,E1 -17919.621,E2 -17919.621} C_VEL
LIN {X 0,Y 285.01,Z 487.313,A -85,B 0,C 180,E1 -17920.389,E2 -17920.389} C_VEL
LIN {X 0,Y 285.746,Z 473.925,A -85,B 0,C 180,E1 -17920.855,E2 -17920.855} C_VEL
LIN {X 0,Y 288.503,Z 387.671,A -85,B 0,C 180,E1 -17922.993,E2 -17922.993} C_VEL
LIN {X 0,Y 280.711,Z 367.647,A -85,B 0,C 180,E1 -17924.351,E2 -17924.351} C_VEL
LIN {X 0,Y 274.949,Z 355.021,A -85,B 0,C 180,E1 -17925.346,E2 -17925.346} C_VEL
LIN {X 0,Y 270.496,Z 346.282,A -85,B 0,C 180,E1 -17926.116,E2 -17926.116} C_VEL
LIN {X 0,Y 270.314,Z 345.442,A -85,B 0,C 180,E1 -17926.233,E2 -17926.233} C_VEL
LIN {X 0,Y 270.27,Z 345.449,A -85,B 0,C 180,E1 -17930.591,E2 -17930.591} C_VEL
LIN {X 0,Y 270.223,Z 345.451,A -85,B 0,C 180,E1 -17934.592,E2 -17934.592} C_VEL
LIN {X 0,Y 270.192,Z 345.452,A -85,B 0,C 180,E1 -17937.919,E2 -17937.919} C_VEL
LIN {X 0,Y 270.168,Z 345.456,A -85,B 0,C 180,E1 -17941.352,E2 -17941.352} C_VEL
LIN {X 0,Y 270.198,Z 345.45,A -85,B 0,C 180,E1 -17944.907,E2 -17944.907} C_VEL
LIN {X 0,Y 270.198,Z 345.45,A -85,B 0,C 180,E1 -17948.712,E2 -17948.712} C_VEL
LIN {X 0,Y 270.148,Z 345.447,A -85,B 0,C 180,E1 -17953.246,E2 -17953.246} C_VEL
LIN {X 0,Y 270.151,Z 345.455,A -85,B 0,C 180,E1 -17957.439,E2 -17957.439} C_VEL
LIN {X 0,Y 270.153,Z 345.45,A -85,B 0,C 180,E1 -17961.366,E2 -17961.366} C_VEL
LIN {X 0,Y 270.199,Z 345.438,A -85,B 0,C 180,E1 -17965.095,E2 -17965.095} C_VEL
LIN {X 0,Y 270.173,Z 345.455,A -85,B 0,C 180,E1 -17969.142,E2 -17969.142} C_VEL
LIN {X 0,Y 270.19,Z 345.45,A -85,B 0,C 180,E1 -17972.178,E2 -17972.178} C_VEL
LIN {X 0,Y 270.184,Z 345.453,A -85,B 0,C 180,E1 -17975.565,E2 -17975.565} C_VEL
LIN {X 0,Y 270.224,Z 345.449,A -85,B 0,C 180,E1 -17980.239,E2 -17980.239} C_VEL
LIN {X 0,Y 270.217,Z 345.449,A -85,B 0,C 180,E1 -17980.361,E2 -17980.361} C_VEL
LIN {X 0,Y 269.515,Z 345.537,A -85,B 0,C 180,E1 -17981.607,E2 -17981.607} C_VEL
LIN {X 0,Y 266.678,Z 345.887,A -85,B 0,C 180,E1 -17983.638,E2 -17983.638} C_VEL
LIN {X 0,Y 264.313,Z 346.173,A -85,B 0,C 180,E1 -17985.289,E2 -17985.289} C_VEL
LIN {X 0,Y 263.327,Z 346.284,A -85,B 0,C 180,E1 -17986.568,E2 -17986.568} C_VEL
LIN {X 0,Y 263.261,Z 346.29,A -85,B 0,C 180,E1 -17987.001,E2 -17987.001} C_VEL
LIN {X 0,Y 263.476,Z 346.284,A -85,B 0,C 180,E1 -17990.791,E2 -17990.791} C_VEL
LIN {X 0,Y 263.489,Z 346.289,A -85,B 0,C 180,E1 -17993.876,E2 -17993.876} C_VEL
LIN {X 0,Y 263.747,Z 346.235,A -85,B 0,C 180,E1 -17998.474,E2 -17998.474} C_VEL
LIN {X 0,Y 263.745,Z 346.241,A -85,B 0,C 180,E1 -18001.527,E2 -18001.527} C_VEL
LIN {X 0,Y 263.538,Z 346.28,A -85,B 0,C 180,E1 -18007.663,E2 -18007.663} C_VEL
LIN {X 0,Y 263.355,Z 346.303,A -85,B 0,C 180,E1 -18010.767,E2 -18010.767} C_VEL
LIN {X 0,Y 263.356,Z 346.303,A -85,B 0,C 180,E1 -18015.478,E2 -18015.478} C_VEL
LIN {X 0,Y 263.27,Z 346.311,A -85,B 0,C 180,E1 -18020.307,E2 -18020.307} C_VEL
LIN {X 0,Y 263.213,Z 346.317,A -85,B 0,C 180,E1 -18025.291,E2 -18025.291} C_VEL
LIN {X 0,Y 263.171,Z 346.324,A -85,B 0,C 180,E1 -18028.731,E2 -18028.731} C_VEL
LIN {X 0,Y 263.138,Z 346.33,A -85,B 0,C 180,E1 -18032.288,E2 -18032.288} C_VEL
LIN {X 0,Y 263.187,Z 346.324,A -85,B 0,C 180,E1 -18036.763,E2 -18036.763} C_VEL
LIN {X 0,Y 263.13,Z 346.333,A -85,B 0,C 180,E1 -18041.593,E2 -18041.593} C_VEL
LIN {X 0,Y 263.133,Z 346.33,A -85,B 0,C 180,E1 -18046.017,E2 -18046.017} C_VEL
LIN {X 0,Y 263.164,Z 346.401,A -85,B 0,C 180,E1 -18050.505,E2 -18050.505} C_VEL
LIN {X 0,Y 265.644,Z 356.384,A -85,B 0,C 180,E1 -18053.949,E2 -18053.949} C_VEL
LIN {X 0,Y 266.607,Z 360.73,A -85,B 0,C 180,E1 -18055.345,E2 -18055.345} C_VEL
LIN {X 0,Y 275.278,Z 382.028,A -85,B 0,C 180,E1 -18056.964,E2 -18056.964} C_VEL
LIN {X 0,Y 277.644,Z 388.695,A -85,B 0,C 180,E1 -18057.411,E2 -18057.411} C_VEL
LIN {X 0,Y 281.489,Z 415.729,A -85,B 0,C 180,E1 -18058.58,E2 -18058.58} C_VEL
LIN {X 0,Y 278.566,Z 499.765,A -85,B 0,C 180,E1 -18060.736,E2 -18060.736} C_VEL
LIN {X 0,Y 277.444,Z 514.221,A -85,B 0,C 180,E1 -18061.384,E2 -18061.384} C_VEL
LIN {X 0,Y 275.885,Z 528.145,A -85,B 0,C 180,E1 -18062.295,E2 -18062.295} C_VEL
LIN {X 0,Y 273.953,Z 542.038,A -85,B 0,C 180,E1 -18063.528,E2 -18063.528} C_VEL
LIN {X 0,Y 272.104,Z 554.63,A -85,B 0,C 180,E1 -18064.99,E2 -18064.99} C_VEL
LIN {X 0,Y 270.262,Z 564.758,A -85,B 0,C 180,E1 -18066.432,E2 -18066.432} C_VEL
LIN {X 0,Y 268.33,Z 574.443,A -85,B 0,C 180,E1 -18068.084,E2 -18068.084} C_VEL
LIN {X 0,Y 266.274,Z 585.221,A -85,B 0,C 180,E1 -18070.334,E2 -18070.334} C_VEL
LIN {X 0,Y 264.632,Z 594.104,A -85,B 0,C 180,E1 -18072.615,E2 -18072.615} C_VEL
LIN {X 0,Y 263.163,Z 602.601,A -85,B 0,C 180,E1 -18075.302,E2 -18075.302} C_VEL
LIN {X 0,Y 262.184,Z 608.493,A -85,B 0,C 180,E1 -18077.616,E2 -18077.616} C_VEL
LIN {X 0,Y 261.582,Z 613.334,A -85,B 0,C 180,E1 -18079.941,E2 -18079.941} C_VEL
LIN {X 0,Y 261.29,Z 617.241,A -85,B 0,C 180,E1 -18082.27,E2 -18082.27} C_VEL
LIN {X 0,Y 261.102,Z 621.027,A -85,B 0,C 180,E1 -18085.367,E2 -18085.367} C_VEL
LIN {X 0,Y 261.143,Z 622.374,A -85,B 0,C 180,E1 -18086.913,E2 -18086.913} C_VEL
LIN {X 0,Y 261.171,Z 623.367,A -85,B 0,C 180,E1 -18088.457,E2 -18088.457} C_VEL
LIN {X 0,Y 261.179,Z 624.014,A -85,B 0,C 180,E1 -18089.999,E2 -18089.999} C_VEL
LIN {X 0,Y 261.099,Z 624.288,A -85,B 0,C 180,E1 -18093.085,E2 -18093.085} C_VEL
LIN {X 0,Y 261.143,Z 623.228,A -85,B 0,C 180,E1 -18096.178,E2 -18096.178} C_VEL
LIN {X 0,Y 261.509,Z 620.837,A -85,B 0,C 180,E1 -18099.278,E2 -18099.278} C_VEL
LIN {X 0,Y 262.368,Z 617.067,A -85,B 0,C 180,E1 -18102.373,E2 -18102.373} C_VEL
LIN {X 0,Y 264.005,Z 611.825,A -85,B 0,C 180,E1 -18105.437,E2 -18105.437} C_VEL
LIN {X 0,Y 265.659,Z 606.436,A -85,B 0,C 180,E1 -18107.863,E2 -18107.863} C_VEL
LIN {X 0,Y 268.312,Z 598.503,A -85,B 0,C 180,E1 -18110.707,E2 -18110.707} C_VEL
LIN {X 0,Y 270.91,Z 590.813,A -85,B 0,C 180,E1 -18112.899,E2 -18112.899} C_VEL
LIN {X 0,Y 273.939,Z 581.627,A -85,B 0,C 180,E1 -18115.042,E2 -18115.042} C_VEL
LIN {X 0,Y 277.338,Z 570.5,A -85,B 0,C 180,E1 -18117.136,E2 -18117.136} C_VEL
LIN {X 0,Y 280.436,Z 559.212,A -85,B 0,C 180,E1 -18118.842,E2 -18118.842} C_VEL
LIN {X 0,Y 283.177,Z 548.33,A -85,B 0,C 180,E1 -18120.169,E2 -18120.169} C_VEL
LIN {X 0,Y 285.605,Z 536.741,A -85,B 0,C 180,E1 -18121.319,E2 -18121.319} C_VEL
LIN {X 0,Y 288.19,Z 522.954,A -85,B 0,C 180,E1 -18122.341,E2 -18122.341} C_VEL
LIN {X 0,Y 290.084,Z 509.351,A -85,B 0,C 180,E1 -18123.083,E2 -18123.083} C_VEL
LIN {X 0,Y 291.328,Z 495.618,A -85,B 0,C 180,E1 -18123.595,E2 -18123.595} C_VEL
LIN {X 0,Y 294.883,Z 418.672,A -85,B 0,C 180,E1 -18125.509,E2 -18125.509} C_VEL
LIN {X 0,Y 293.054,Z 406.738,A -85,B 0,C 180,E1 -18126.212,E2 -18126.212} C_VEL
LIN {X 0,Y 286.088,Z 391.465,A -85,B 0,C 180,E1 -18127.997,E2 -18127.997} C_VEL
LIN {X 0,Y 279.096,Z 378.422,A -85,B 0,C 180,E1 -18129.874,E2 -18129.874} C_VEL
LIN {X 0,Y 273.449,Z 368.781,A -85,B 0,C 180,E1 -18131.475,E2 -18131.475} C_VEL
LIN {X 0,Y 270.082,Z 363.382,A -85,B 0,C 180,E1 -18132.477,E2 -18132.477} C_VEL
LIN {X 0,Y 267.199,Z 358.798,A -85,B 0,C 180,E1 -18133.376,E2 -18133.376} C_VEL
LIN {X 0,Y 266.872,Z 357.975,A -85,B 0,C 180,E1 -18133.666,E2 -18133.666} C_VEL
LIN {X 0,Y 264.483,Z 350.688,A -85,B 0,C 180,E1 -18137.344,E2 -18137.344} C_VEL
LIN {X 0,Y 263.116,Z 346.312,A -85,B 0,C 180,E1 -18139.754,E2 -18139.754} C_VEL
LIN {X 0,Y 263.182,Z 346.321,A -85,B 0,C 180,E1 -18144.021,E2 -18144.021} C_VEL
LIN {X 0,Y 263.128,Z 346.327,A -85,B 0,C 180,E1 -18147.711,E2 -18147.711} C_VEL
LIN {X 0,Y 263.196,Z 346.325,A -85,B 0,C 180,E1 -18151.782,E2 -18151.782} C_VEL
LIN {X 0,Y 263.22,Z 346.323,A -85,B 0,C 180,E1 -18155.199,E2 -18155.199} C_VEL
LIN {X 0,Y 263.257,Z 346.315,A -85,B 0,C 180,E1 -18159.692,E2 -18159.692} C_VEL
LIN {X 0,Y 263.344,Z 346.296,A -85,B 0,C 180,E1 -18164.521,E2 -18164.521} C_VEL
LIN {X 0,Y 263.367,Z 346.292,A -85,B 0,C 180,E1 -18169.234,E2 -18169.234} C_VEL
LIN {X 0,Y 263.565,Z 346.27,A -85,B 0,C 180,E1 -18172.338,E2 -18172.338} C_VEL
LIN {X 0,Y 263.732,Z 346.254,A -85,B 0,C 180,E1 -18178.472,E2 -18178.472} C_VEL
LIN {X 0,Y 263.726,Z 346.248,A -85,B 0,C 180,E1 -18181.527,E2 -18181.527} C_VEL
LIN {X 0,Y 263.516,Z 346.284,A -85,B 0,C 180,E1 -18187.663,E2 -18187.663} C_VEL
LIN {X 0,Y 263.34,Z 346.308,A -85,B 0,C 180,E1 -18190.766,E2 -18190.766} C_VEL
LIN {X 0,Y 263.301,Z 346.306,A -85,B 0,C 180,E1 -18195.48,E2 -18195.48} C_VEL
LIN {X 0,Y 263.227,Z 346.319,A -85,B 0,C 180,E1 -18200.309,E2 -18200.309} C_VEL
LIN {X 0,Y 263.159,Z 346.326,A -85,B 0,C 180,E1 -18205.296,E2 -18205.296} C_VEL
LIN {X 0,Y 263.195,Z 346.42,A -85,B 0,C 180,E1 -18207.617,E2 -18207.617} C_VEL
LIN {X 0,Y 264.023,Z 348.917,A -85,B 0,C 180,E1 -18207.948,E2 -18207.948} C_VEL
LIN {X 0,Y 265.856,Z 351.057,A -85,B 0,C 180,E1 -18208.521,E2 -18208.521} C_VEL
LIN {X 0,Y 266.761,Z 351.943,A -85,B 0,C 180,E1 -18208.791,E2 -18208.791} C_VEL
LIN {X 0,Y 268.857,Z 355.236,A -85,B 0,C 180,E1 -18209.456,E2 -18209.456} C_VEL
LIN {X 0,Y 270.391,Z 357.023,A -85,B 0,C 180,E1 -18209.905,E2 -18209.905} C_VEL
LIN {X 0,Y 273.149,Z 360.736,A -85,B 0,C 180,E1 -18210.704,E2 -18210.704} C_VEL
LIN {X 0,Y 279.556,Z 370.471,A -85,B 0,C 180,E1 -18212.49,E2 -18212.49} C_VEL
LIN {X 0,Y 285.85,Z 381.151,A -85,B 0,C 180,E1 -18214.156,E2 -18214.156} C_VEL
LIN {X 0,Y 292.677,Z 394.356,A -85,B 0,C 180,E1 -18215.877,E2 -18215.877} C_VEL
LIN {X 0,Y 295.686,Z 400.867,A -85,B 0,C 180,E1 -18216.614,E2 -18216.614} C_VEL
LIN {X 0,Y 291.867,Z 480.729,A -85,B 0,C 180,E1 -18218.598,E2 -18218.598} C_VEL
LIN {X 0,Y 290.551,Z 495.163,A -85,B 0,C 180,E1 -18219.212,E2 -18219.212} C_VEL
LIN {X 0,Y 288.653,Z 508.927,A -85,B 0,C 180,E1 -18220.058,E2 -18220.058} C_VEL
LIN {X 0,Y 286.517,Z 521.74,A -85,B 0,C 180,E1 -18221.137,E2 -18221.137} C_VEL
LIN {X 0,Y 283.734,Z 534.763,A -85,B 0,C 180,E1 -18222.535,E2 -18222.535} C_VEL
LIN {X 0,Y 280.824,Z 546.393,A -85,B 0,C 180,E1 -18224.111,E2 -18224.111} C_VEL
LIN {X 0,Y 277.787,Z 557.137,A -85,B 0,C 180,E1 -18225.915,E2 -18225.915} C_VEL
LIN {X 0,Y 274.876,Z 566.53,A -85,B 0,C 180,E1 -18227.856,E2 -18227.856} C_VEL
LIN {X 0,Y 271.796,Z 575.738,A -85,B 0,C 180,E1 -18230.193,E2 -18230.193} C_VEL
LIN {X 0,Y 269.078,Z 583.382,A -85,B 0,C 180,E1 -18232.61,E2 -18232.61} C_VEL
LIN {X 0,Y 266.517,Z 590.465,A -85,B 0,C 180,E1 -18235.464,E2 -18235.464} C_VEL
LIN {X 0,Y 264.617,Z 595.696,A -85,B 0,C 180,E1 -18238.199,E2 -18238.199} C_VEL
LIN {X 0,Y 263.026,Z 599.995,A -85,B 0,C 180,E1 -18241.254,E2 -18241.254} C_VEL
LIN {X 0,Y 262.388,Z 601.721,A -85,B 0,C 180,E1 -18242.915,E2 -18242.915} C_VEL
LIN {X 0,Y 261.471,Z 603.995,A -85,B 0,C 180,E1 -18246.225,E2 -18246.225} C_VEL
LIN {X 0,Y 260.979,Z 604.767,A -85,B 0,C 180,E1 -18249.509,E2 -18249.509} C_VEL
LIN {X 0,Y 260.9,Z 604.603,A -85,B 0,C 180,E1 -18251.142,E2 -18251.142} C_VEL
LIN {X 0,Y 260.867,Z 603.172,A -85,B 0,C 180,E1 -18254.372,E2 -18254.372} C_VEL
LIN {X 0,Y 261.049,Z 601.909,A -85,B 0,C 180,E1 -18255.979,E2 -18255.979} C_VEL
LIN {X 0,Y 261.525,Z 598.301,A -85,B 0,C 180,E1 -18259.159,E2 -18259.159} C_VEL
LIN {X 0,Y 262.316,Z 593.162,A -85,B 0,C 180,E1 -18262.303,E2 -18262.303} C_VEL
LIN {X 0,Y 263.149,Z 588.19,A -85,B 0,C 180,E1 -18264.638,E2 -18264.638} C_VEL
LIN {X 0,Y 264.46,Z 581.04,A -85,B 0,C 180,E1 -18267.336,E2 -18267.336} C_VEL
LIN {X 0,Y 266.233,Z 572.183,A -85,B 0,C 180,E1 -18270.001,E2 -18270.001} C_VEL
LIN {X 0,Y 268.042,Z 562.919,A -85,B 0,C 180,E1 -18272.255,E2 -18272.255} C_VEL
LIN {X 0,Y 269.944,Z 552.698,A -85,B 0,C 180,E1 -18274.294,E2 -18274.294} C_VEL
LIN {X 0,Y 271.98,Z 541.412,A -85,B 0,C 180,E1 -18276.12,E2 -18276.12} C_VEL
LIN {X 0,Y 274.014,Z 528.92,A -85,B 0,C 180,E1 -18277.74,E2 -18277.74} C_VEL
LIN {X 0,Y 275.698,Z 516.892,A -85,B 0,C 180,E1 -18278.984,E2 -18278.984} C_VEL
LIN {X 0,Y 277.164,Z 503.759,A -85,B 0,C 180,E1 -18280.041,E2 -18280.041} C_VEL
LIN {X 0,Y 278.353,Z 489.597,A -85,B 0,C 180,E1 -18280.871,E2 -18280.871} C_VEL
LIN {X 0,Y 279.166,Z 476.016,A -85,B 0,C 180,E1 -18281.39,E2 -18281.39} C_VEL
LIN {X 0,Y 282.165,Z 389.57,A -85,B 0,C 180,E1 -18283.572,E2 -18283.572} C_VEL
LIN {X 0,Y 274.295,Z 369.358,A -85,B 0,C 180,E1 -18284.992,E2 -18284.992} C_VEL
LIN {X 0,Y 269.11,Z 358.151,A -85,B 0,C 180,E1 -18285.916,E2 -18285.916} C_VEL
LIN {X 0,Y 263.546,Z 347.679,A -85,B 0,C 180,E1 -18286.906,E2 -18286.906} C_VEL
LIN {X 0,Y 263.246,Z 346.325,A -85,B 0,C 180,E1 -18287.003,E2 -18287.003} C_VEL
LIN {X 0,Y 263.198,Z 346.331,A -85,B 0,C 180,E1 -18290.841,E2 -18290.841} C_VEL
LIN {X 0,Y 263.166,Z 346.33,A -85,B 0,C 180,E1 -18295.297,E2 -18295.297} C_VEL
LIN {X 0,Y 263.122,Z 346.335,A -85,B 0,C 180,E1 -18298.738,E2 -18298.738} C_VEL
LIN {X 0,Y 263.126,Z 346.332,A -85,B 0,C 180,E1 -18302.291,E2 -18302.291} C_VEL
LIN {X 0,Y 263.176,Z 346.317,A -85,B 0,C 180,E1 -18306.762,E2 -18306.762} C_VEL
LIN {X 0,Y 263.092,Z 346.337,A -85,B 0,C 180,E1 -18309.876,E2 -18309.876} C_VEL
LIN {X 0,Y 263.077,Z 346.325,A -85,B 0,C 180,E1 -18313.995,E2 -18313.995} C_VEL
LIN {X 0,Y 263.074,Z 346.339,A -85,B 0,C 180,E1 -18318.42,E2 -18318.42} C_VEL
LIN {X 0,Y 263.105,Z 346.326,A -85,B 0,C 180,E1 -18322.095,E2 -18322.095} C_VEL
LIN {X 0,Y 263.153,Z 346.317,A -85,B 0,C 180,E1 -18325.887,E2 -18325.887} C_VEL
LIN {X 0,Y 263.111,Z 346.334,A -85,B 0,C 180,E1 -18329.502,E2 -18329.502} C_VEL
LIN {X 0,Y 263.114,Z 346.332,A -85,B 0,C 180,E1 -18332.995,E2 -18332.995} C_VEL
LIN {X 0,Y 263.118,Z 346.335,A -85,B 0,C 180,E1 -18336.381,E2 -18336.381} C_VEL
LIN {X 0,Y 263.166,Z 346.322,A -85,B 0,C 180,E1 -18340.348,E2 -18340.348} C_VEL
LIN {X 0,Y 263.294,Z 346.303,A -85,B 0,C 180,E1 -18344.519,E2 -18344.519} C_VEL
LIN {X 0,Y 263.261,Z 346.29,A -85,B 0,C 180,E1 -18347.001,E2 -18347.001} C_VEL
LIN {X 0,Y 262.678,Z 346.367,A -85,B 0,C 180,E1 -18348.279,E2 -18348.279} C_VEL
LIN {X 0,Y 260.018,Z 346.713,A -85,B 0,C 180,E1 -18350.367,E2 -18350.367} C_VEL
LIN {X 0,Y 256.844,Z 347.119,A -85,B 0,C 180,E1 -18352.934,E2 -18352.934} C_VEL
LIN {X 0,Y 256.445,Z 347.164,A -85,B 0,C 180,E1 -18353.82,E2 -18353.82} C_VEL
LIN {X 0,Y 256.709,Z 347.111,A -85,B 0,C 180,E1 -18358.432,E2 -18358.432} C_VEL
LIN {X 0,Y 256.707,Z 347.117,A -85,B 0,C 180,E1 -18361.569,E2 -18361.569} C_VEL
LIN {X 0,Y 256.467,Z 347.162,A -85,B 0,C 180,E1 -18366.294,E2 -18366.294} C_VEL
LIN {X 0,Y 256.432,Z 347.163,A -85,B 0,C 180,E1 -18369.465,E2 -18369.465} C_VEL
LIN {X 0,Y 256.26,Z 347.186,A -85,B 0,C 180,E1 -18374.29,E2 -18374.29} C_VEL
LIN {X 0,Y 256.216,Z 347.195,A -85,B 0,C 180,E1 -18377.562,E2 -18377.562} C_VEL
LIN {X 0,Y 256.165,Z 347.197,A -85,B 0,C 180,E1 -18381.121,E2 -18381.121} C_VEL
LIN {X 0,Y 256.194,Z 347.191,A -85,B 0,C 180,E1 -18385.138,E2 -18385.138} C_VEL
LIN {X 0,Y 256.109,Z 347.203,A -85,B 0,C 180,E1 -18389.601,E2 -18389.601} C_VEL
LIN {X 0,Y 256.073,Z 347.21,A -85,B 0,C 180,E1 -18393.293,E2 -18393.293} C_VEL
LIN {X 0,Y 256.119,Z 347.199,A -85,B 0,C 180,E1 -18397.27,E2 -18397.27} C_VEL
LIN {X 0,Y 256.06,Z 347.216,A -85,B 0,C 180,E1 -18401.203,E2 -18401.203} C_VEL
LIN {X 0,Y 256.067,Z 347.212,A -85,B 0,C 180,E1 -18405.529,E2 -18405.529} C_VEL
LIN {X 0,Y 256.094,Z 347.3,A -85,B 0,C 180,E1 -18409.836,E2 -18409.836} C_VEL
LIN {X 0,Y 258.778,Z 358.027,A -85,B 0,C 180,E1 -18413.664,E2 -18413.664} C_VEL
LIN {X 0,Y 259.328,Z 360.389,A -85,B 0,C 180,E1 -18414.444,E2 -18414.444} C_VEL
LIN {X 0,Y 268.609,Z 382.849,A -85,B 0,C 180,E1 -18416.252,E2 -18416.252} C_VEL
LIN {X 0,Y 271.507,Z 390.875,A -85,B 0,C 180,E1 -18416.816,E2 -18416.816} C_VEL
LIN {X 0,Y 275.078,Z 417.012,A -85,B 0,C 180,E1 -18417.97,E2 -18417.97} C_VEL
LIN {X 0,Y 272.155,Z 498.298,A -85,B 0,C 180,E1 -18420.084,E2 -18420.084} C_VEL
LIN {X 0,Y 271.087,Z 512.436,A -85,B 0,C 180,E1 -18420.702,E2 -18420.702} C_VEL
LIN {X 0,Y 269.614,Z 526.206,A -85,B 0,C 180,E1 -18421.592,E2 -18421.592} C_VEL
LIN {X 0,Y 267.87,Z 538.679,A -85,B 0,C 180,E1 -18422.667,E2 -18422.667} C_VEL
LIN {X 0,Y 265.986,Z 550.665,A -85,B 0,C 180,E1 -18423.993,E2 -18423.993} C_VEL
LIN {X 0,Y 264.066,Z 561.222,A -85,B 0,C 180,E1 -18425.426,E2 -18425.426} C_VEL
LIN {X 0,Y 261.937,Z 572.476,A -85,B 0,C 180,E1 -18427.312,E2 -18427.312} C_VEL
LIN {X 0,Y 259.85,Z 582.703,A -85,B 0,C 180,E1 -18429.413,E2 -18429.413} C_VEL
LIN {X 0,Y 258.049,Z 591.964,A -85,B 0,C 180,E1 -18431.746,E2 -18431.746} C_VEL
LIN {X 0,Y 256.668,Z 599.661,A -85,B 0,C 180,E1 -18434.107,E2 -18434.107} C_VEL
LIN {X 0,Y 255.558,Z 606.06,A -85,B 0,C 180,E1 -18436.48,E2 -18436.48} C_VEL
LIN {X 0,Y 254.704,Z 611.296,A -85,B 0,C 180,E1 -18438.862,E2 -18438.862} C_VEL
LIN {X 0,Y 254.304,Z 615.537,A -85,B 0,C 180,E1 -18441.256,E2 -18441.256} C_VEL
LIN {X 0,Y 254.074,Z 618.891,A -85,B 0,C 180,E1 -18443.646,E2 -18443.646} C_VEL
LIN {X 0,Y 254.055,Z 622.005,A -85,B 0,C 180,E1 -18446.827,E2 -18446.827} C_VEL
LIN {X 0,Y 254.097,Z 623.028,A -85,B 0,C 180,E1 -18448.414,E2 -18448.414} C_VEL
LIN {X 0,Y 254.104,Z 623.703,A -85,B 0,C 180,E1 -18449.999,E2 -18449.999} C_VEL
LIN {X 0,Y 254.075,Z 624.036,A -85,B 0,C 180,E1 -18451.584,E2 -18451.584} C_VEL
LIN {X 0,Y 253.974,Z 623.694,A -85,B 0,C 180,E1 -18454.76,E2 -18454.76} C_VEL
LIN {X 0,Y 254.214,Z 622.03,A -85,B 0,C 180,E1 -18457.944,E2 -18457.944} C_VEL
LIN {X 0,Y 254.892,Z 619.023,A -85,B 0,C 180,E1 -18461.127,E2 -18461.127} C_VEL
LIN {X 0,Y 256.228,Z 614.6,A -85,B 0,C 180,E1 -18464.29,E2 -18464.29} C_VEL
LIN {X 0,Y 258.201,Z 608.641,A -85,B 0,C 180,E1 -18467.421,E2 -18467.421} C_VEL
LIN {X 0,Y 260.455,Z 601.982,A -85,B 0,C 180,E1 -18470.122,E2 -18470.122} C_VEL
LIN {X 0,Y 263.394,Z 593.751,A -85,B 0,C 180,E1 -18472.76,E2 -18472.76} C_VEL
LIN {X 0,Y 266.382,Z 585.206,A -85,B 0,C 180,E1 -18474.967,E2 -18474.967} C_VEL
LIN {X 0,Y 269.863,Z 574.897,A -85,B 0,C 180,E1 -18477.111,E2 -18477.111} C_VEL
LIN {X 0,Y 273.062,Z 564.095,A -85,B 0,C 180,E1 -18478.944,E2 -18478.944} C_VEL
LIN {X 0,Y 276.332,Z 552.053,A -85,B 0,C 180,E1 -18480.573,E2 -18480.573} C_VEL
LIN {X 0,Y 279.267,Z 539.616,A -85,B 0,C 180,E1 -18481.901,E2 -18481.901} C_VEL
LIN {X 0,Y 282.09,Z 525.724,A -85,B 0,C 180,E1 -18483.022,E2 -18483.022} C_VEL
LIN {X 0,Y 284.235,Z 511.759,A -85,B 0,C 180,E1 -18483.854,E2 -18483.854} C_VEL
LIN {X 0,Y 285.8,Z 497.037,A -85,B 0,C 180,E1 -18484.441,E2 -18484.441} C_VEL
LIN {X 0,Y 289.547,Z 420.029,A -85,B 0,C 180,E1 -18486.386,E2 -18486.386} C_VEL
LIN {X 0,Y 287.939,Z 409.696,A -85,B 0,C 180,E1 -18487.023,E2 -18487.023} C_VEL
LIN {X 0,Y 281.703,Z 395.829,A -85,B 0,C 180,E1 -18488.707,E2 -18488.707} C_VEL
LIN {X 0,Y 275.204,Z 383.46,A -85,B 0,C 180,E1 -18490.523,E2 -18490.523} C_VEL
LIN {X 0,Y 269.451,Z 373.578,A -85,B 0,C 180,E1 -18492.217,E2 -18492.217} C_VEL
LIN {X 0,Y 266.065,Z 368.113,A -85,B 0,C 180,E1 -18493.272,E2 -18493.272} C_VEL
LIN {X 0,Y 262.845,Z 363.132,A -85,B 0,C 180,E1 -18494.315,E2 -18494.315} C_VEL
LIN {X 0,Y 259.753,Z 358.396,A -85,B 0,C 180,E1 -18495.362,E2 -18495.362} C_VEL
LIN {X 0,Y 259.38,Z 357.362,A -85,B 0,C 180,E1 -18495.756,E2 -18495.756} C_VEL
LIN {X 0,Y 257.405,Z 351.34,A -85,B 0,C 180,E1 -18499.059,E2 -18499.059} C_VEL
LIN {X 0,Y 256.095,Z 347.192,A -85,B 0,C 180,E1 -18501.614,E2 -18501.614} C_VEL
LIN {X 0,Y 256.118,Z 347.207,A -85,B 0,C 180,E1 -18505.404,E2 -18505.404} C_VEL
LIN {X 0,Y 256.087,Z 347.211,A -85,B 0,C 180,E1 -18508.571,E2 -18508.571} C_VEL
LIN {X 0,Y 256.136,Z 347.204,A -85,B 0,C 180,E1 -18512.195,E2 -18512.195} C_VEL
LIN {X 0,Y 256.161,Z 347.202,A -85,B 0,C 180,E1 -18515.698,E2 -18515.698} C_VEL
LIN {X 0,Y 256.161,Z 347.202,A -85,B 0,C 180,E1 -18519.104,E2 -18519.104} C_VEL
LIN {X 0,Y 256.293,Z 347.176,A -85,B 0,C 180,E1 -18524.084,E2 -18524.084} C_VEL
LIN {X 0,Y 256.303,Z 347.171,A -85,B 0,C 180,E1 -18528.933,E2 -18528.933} C_VEL
LIN {X 0,Y 256.532,Z 347.148,A -85,B 0,C 180,E1 -18532.126,E2 -18532.126} C_VEL
LIN {X 0,Y 256.694,Z 347.13,A -85,B 0,C 180,E1 -18538.431,E2 -18538.431} C_VEL
LIN {X 0,Y 256.689,Z 347.125,A -85,B 0,C 180,E1 -18541.568,E2 -18541.568} C_VEL
LIN {X 0,Y 256.434,Z 347.16,A -85,B 0,C 180,E1 -18546.565,E2 -18546.565} C_VEL
LIN {X 0,Y 256.419,Z 347.16,A -85,B 0,C 180,E1 -18549.465,E2 -18549.465} C_VEL
LIN {X 0,Y 256.223,Z 347.195,A -85,B 0,C 180,E1 -18554.291,E2 -18554.291} C_VEL
LIN {X 0,Y 256.159,Z 347.202,A -85,B 0,C 180,E1 -18557.565,E2 -18557.565} C_VEL
LIN {X 0,Y 256.133,Z 347.205,A -85,B 0,C 180,E1 -18561.11,E2 -18561.11} C_VEL
LIN {X 0,Y 256.109,Z 347.335,A -85,B 0,C 180,E1 -18565.629,E2 -18565.629} C_VEL
LIN {X 0,Y 256.968,Z 349.865,A -85,B 0,C 180,E1 -18566.004,E2 -18566.004} C_VEL
LIN {X 0,Y 259.011,Z 352.116,A -85,B 0,C 180,E1 -18566.705,E2 -18566.705} C_VEL
LIN {X 0,Y 259.886,Z 352.846,A -85,B 0,C 180,E1 -18566.988,E2 -18566.988} C_VEL
LIN {X 0,Y 261.794,Z 355.987,A -85,B 0,C 180,E1 -18567.659,E2 -18567.659} C_VEL
LIN {X 0,Y 263.529,Z 357.911,A -85,B 0,C 180,E1 -18568.207,E2 -18568.207} C_VEL
LIN {X 0,Y 266.18,Z 361.57,A -85,B 0,C 180,E1 -18569.049,E2 -18569.049} C_VEL
LIN {X 0,Y 272.919,Z 371.074,A -85,B 0,C 180,E1 -18571.052,E2 -18571.052} C_VEL
LIN {X 0,Y 279.791,Z 382.505,A -85,B 0,C 180,E1 -18572.981,E2 -18572.981} C_VEL
LIN {X 0,Y 286.148,Z 394.512,A -85,B 0,C 180,E1 -18574.683,E2 -18574.683} C_VEL
LIN {X 0,Y 290.307,Z 403.299,A -85,B 0,C 180,E1 -18575.754,E2 -18575.754} C_VEL
LIN {X 0,Y 286.342,Z 481.69,A -85,B 0,C 180,E1 -18577.728,E2 -18577.728} C_VEL
LIN {X 0,Y 284.909,Z 496.4,A -85,B 0,C 180,E1 -18578.378,E2 -18578.378} C_VEL
LIN {X 0,Y 282.951,Z 509.871,A -85,B 0,C 180,E1 -18579.23,E2 -18579.23} C_VEL
LIN {X 0,Y 280.907,Z 521.7,A -85,B 0,C 180,E1 -18580.244,E2 -18580.244} C_VEL
LIN {X 0,Y 278.235,Z 533.93,A -85,B 0,C 180,E1 -18581.559,E2 -18581.559} C_VEL
LIN {X 0,Y 275.347,Z 545.146,A -85,B 0,C 180,E1 -18583.064,E2 -18583.064} C_VEL
LIN {X 0,Y 271.952,Z 556.615,A -85,B 0,C 180,E1 -18584.975,E2 -18584.975} C_VEL
LIN {X 0,Y 268.626,Z 566.971,A -85,B 0,C 180,E1 -18587.141,E2 -18587.141} C_VEL
LIN {X 0,Y 265.356,Z 576.225,A -85,B 0,C 180,E1 -18589.545,E2 -18589.545} C_VEL
LIN {X 0,Y 262.542,Z 583.784,A -85,B 0,C 180,E1 -18592,E2 -18592} C_VEL
LIN {X 0,Y 260.026,Z 590.32,A -85,B 0,C 180,E1 -18594.668,E2 -18594.668} C_VEL
LIN {X 0,Y 257.822,Z 595.975,A -85,B 0,C 180,E1 -18597.674,E2 -18597.674} C_VEL
LIN {X 0,Y 256.288,Z 599.853,A -85,B 0,C 180,E1 -18600.424,E2 -18600.424} C_VEL
LIN {X 0,Y 254.964,Z 603.066,A -85,B 0,C 180,E1 -18603.832,E2 -18603.832} C_VEL
LIN {X 0,Y 254.171,Z 604.732,A -85,B 0,C 180,E1 -18607.227,E2 -18607.227} C_VEL
LIN {X 0,Y 253.826,Z 604.922,A -85,B 0,C 180,E1 -18610.596,E2 -18610.596} C_VEL
LIN {X 0,Y 253.759,Z 603.678,A -85,B 0,C 180,E1 -18613.923,E2 -18613.923} C_VEL
LIN {X 0,Y 253.915,Z 602.465,A -85,B 0,C 180,E1 -18615.635,E2 -18615.635} C_VEL
LIN {X 0,Y 254.351,Z 599.067,A -85,B 0,C 180,E1 -18618.849,E2 -18618.849} C_VEL
LIN {X 0,Y 254.895,Z 595.502,A -85,B 0,C 180,E1 -18621.279,E2 -18621.279} C_VEL
LIN {X 0,Y 255.681,Z 590.982,A -85,B 0,C 180,E1 -18623.689,E2 -18623.689} C_VEL
LIN {X 0,Y 256.833,Z 584.466,A -85,B 0,C 180,E1 -18626.472,E2 -18626.472} C_VEL
LIN {X 0,Y 258.524,Z 576.352,A -85,B 0,C 180,E1 -18629.223,E2 -18629.223} C_VEL
LIN {X 0,Y 260.257,Z 567.868,A -85,B 0,C 180,E1 -18631.549,E2 -18631.549} C_VEL
LIN {X 0,Y 262.249,Z 557.653,A -85,B 0,C 180,E1 -18633.843,E2 -18633.843} C_VEL
LIN {X 0,Y 264.507,Z 546.148,A -85,B 0,C 180,E1 -18635.911,E2 -18635.911} C_VEL
LIN {X 0,Y 266.477,Z 534.723,A -85,B 0,C 180,E1 -18637.579,E2 -18637.579} C_VEL
LIN {X 0,Y 268.398,Z 522.216,A -85,B 0,C 180,E1 -18639.04,E2 -18639.04} C_VEL
LIN {X 0,Y 270.186,Z 508.251,A -85,B 0,C 180,E1 -18640.303,E2 -18640.303} C_VEL
LIN {X 0,Y 271.509,Z 494.223,A -85,B 0,C 180,E1 -18641.243,E2 -18641.243} C_VEL
LIN {X 0,Y 272.558,Z 479.281,A -85,B 0,C 180,E1 -18641.906,E2 -18641.906} C_VEL
LIN {X 0,Y 275.686,Z 390.915,A -85,B 0,C 180,E1 -18644.204,E2 -18644.204} C_VEL
LIN {X 0,Y 268.058,Z 371.451,A -85,B 0,C 180,E1 -18645.633,E2 -18645.633} C_VEL
LIN {X 0,Y 263.043,Z 360.804,A -85,B 0,C 180,E1 -18646.556,E2 -18646.556} C_VEL
LIN {X 0,Y 257.382,Z 350.362,A -85,B 0,C 180,E1 -18647.601,E2 -18647.601} C_VEL
LIN {X 0,Y 256.334,Z 348.071,A -85,B 0,C 180,E1 -18647.812,E2 -18647.812} C_VEL
LIN {X 0,Y 256.162,Z 347.208,A -85,B 0,C 180,E1 -18647.891,E2 -18647.891} C_VEL
LIN {X 0,Y 256.14,Z 347.21,A -85,B 0,C 180,E1 -18651.111,E2 -18651.111} C_VEL
LIN {X 0,Y 256.132,Z 347.207,A -85,B 0,C 180,E1 -18655.113,E2 -18655.113} C_VEL
LIN {X 0,Y 256.042,Z 347.216,A -85,B 0,C 180,E1 -18659.61,E2 -18659.61} C_VEL
LIN {X 0,Y 256.065,Z 347.215,A -85,B 0,C 180,E1 -18663.294,E2 -18663.294} C_VEL
LIN {X 0,Y 256.11,Z 347.198,A -85,B 0,C 180,E1 -18667.27,E2 -18667.27} C_VEL
LIN {X 0,Y 256.019,Z 347.217,A -85,B 0,C 180,E1 -18671.212,E2 -18671.212} C_VEL
LIN {X 0,Y 256.018,Z 347.207,A -85,B 0,C 180,E1 -18675.541,E2 -18675.541} C_VEL
LIN {X 0,Y 256.01,Z 347.221,A -85,B 0,C 180,E1 -18678.789,E2 -18678.789} C_VEL
LIN {X 0,Y 256.1,Z 347.188,A -85,B 0,C 180,E1 -18682.863,E2 -18682.863} C_VEL
LIN {X 0,Y 256.067,Z 347.205,A -85,B 0,C 180,E1 -18686.708,E2 -18686.708} C_VEL
LIN {X 0,Y 256.043,Z 347.217,A -85,B 0,C 180,E1 -18690.392,E2 -18690.392} C_VEL
LIN {X 0,Y 256.068,Z 347.21,A -85,B 0,C 180,E1 -18693.952,E2 -18693.952} C_VEL
LIN {X 0,Y 256.06,Z 347.209,A -85,B 0,C 180,E1 -18697.403,E2 -18697.403} C_VEL
LIN {X 0,Y 256.112,Z 347.207,A -85,B 0,C 180,E1 -18700.775,E2 -18700.775} C_VEL
LIN {X 0,Y 256.217,Z 347.187,A -85,B 0,C 180,E1 -18704.08,E2 -18704.08} C_VEL
LIN {X 0,Y 256.278,Z 347.168,A -85,B 0,C 180,E1 -18708.933,E2 -18708.933} C_VEL
LIN {X 0,Y 256.473,Z 347.16,A -85,B 0,C 180,E1 -18712.126,E2 -18712.126} C_VEL
LIN {X 0,Y 256.445,Z 347.164,A -85,B 0,C 180,E1 -18713.82,E2 -18713.82} C_VEL
LIN {X 0,Y 255.691,Z 347.257,A -85,B 0,C 180,E1 -18715.133,E2 -18715.133} C_VEL
LIN {X 0,Y 252.961,Z 347.589,A -85,B 0,C 180,E1 -18717.282,E2 -18717.282} C_VEL
LIN {X 0,Y 249.965,Z 347.946,A -85,B 0,C 180,E1 -18719.924,E2 -18719.924} C_VEL
LIN {X 0,Y 249.664,Z 347.986,A -85,B 0,C 180,E1 -18720.834,E2 -18720.834} C_VEL
LIN {X 0,Y 249.44,Z 348.036,A -85,B 0,C 180,E1 -18726.472,E2 -18726.472} C_VEL
LIN {X 0,Y 249.348,Z 348.047,A -85,B 0,C 180,E1 -18729.737,E2 -18729.737} C_VEL
LIN {X 0,Y 249.21,Z 348.063,A -85,B 0,C 180,E1 -18734.704,E2 -18734.704} C_VEL
LIN {X 0,Y 249.145,Z 348.071,A -85,B 0,C 180,E1 -18738.077,E2 -18738.077} C_VEL
LIN {X 0,Y 249.094,Z 348.08,A -85,B 0,C 180,E1 -18741.518,E2 -18741.518} C_VEL
LIN {X 0,Y 249.136,Z 348.07,A -85,B 0,C 180,E1 -18745.482,E2 -18745.482} C_VEL
LIN {X 0,Y 249.078,Z 348.08,A -85,B 0,C 180,E1 -18748.989,E2 -18748.989} C_VEL
LIN {X 0,Y 249.036,Z 348.086,A -85,B 0,C 180,E1 -18752.426,E2 -18752.426} C_VEL
LIN {X 0,Y 249.053,Z 348.084,A -85,B 0,C 180,E1 -18756.342,E2 -18756.342} C_VEL
LIN {X 0,Y 249.011,Z 348.092,A -85,B 0,C 180,E1 -18760.478,E2 -18760.478} C_VEL
LIN {X 0,Y 249.013,Z 348.092,A -85,B 0,C 180,E1 -18764.878,E2 -18764.878} C_VEL
LIN {X 0,Y 249.062,Z 348.264,A -85,B 0,C 180,E1 -18769.165,E2 -18769.165} C_VEL
LIN {X 0,Y 251.541,Z 358.021,A -85,B 0,C 180,E1 -18772.776,E2 -18772.776} C_VEL
LIN {X 0,Y 251.989,Z 359.982,A -85,B 0,C 180,E1 -18773.474,E2 -18773.474} C_VEL
LIN {X 0,Y 261.192,Z 381.783,A -85,B 0,C 180,E1 -18775.352,E2 -18775.352} C_VEL
LIN {X 0,Y 265.466,Z 393.626,A -85,B 0,C 180,E1 -18776.222,E2 -18776.222} C_VEL
LIN {X 0,Y 268.715,Z 418.143,A -85,B 0,C 180,E1 -18777.33,E2 -18777.33} C_VEL
LIN {X 0,Y 265.644,Z 499.177,A -85,B 0,C 180,E1 -18779.492,E2 -18779.492} C_VEL
LIN {X 0,Y 264.462,Z 513.66,A -85,B 0,C 180,E1 -18780.168,E2 -18780.168} C_VEL
LIN {X 0,Y 262.853,Z 527.611,A -85,B 0,C 180,E1 -18781.121,E2 -18781.121} C_VEL
LIN {X 0,Y 260.912,Z 540.611,A -85,B 0,C 180,E1 -18782.311,E2 -18782.311} C_VEL
LIN {X 0,Y 258.92,Z 553.151,A -85,B 0,C 180,E1 -18783.805,E2 -18783.805} C_VEL
LIN {X 0,Y 256.682,Z 564.829,A -85,B 0,C 180,E1 -18785.534,E2 -18785.534} C_VEL
LIN {X 0,Y 254.237,Z 576.394,A -85,B 0,C 180,E1 -18787.659,E2 -18787.659} C_VEL
LIN {X 0,Y 252.132,Z 586.707,A -85,B 0,C 180,E1 -18790.033,E2 -18790.033} C_VEL
LIN {X 0,Y 250.241,Z 596.135,A -85,B 0,C 180,E1 -18792.726,E2 -18792.726} C_VEL
LIN {X 0,Y 248.908,Z 603.38,A -85,B 0,C 180,E1 -18795.277,E2 -18795.277} C_VEL
LIN {X 0,Y 247.938,Z 609.083,A -85,B 0,C 180,E1 -18797.724,E2 -18797.724} C_VEL
LIN {X 0,Y 247.249,Z 615.038,A -85,B 0,C 180,E1 -18801.004,E2 -18801.004} C_VEL
LIN {X 0,Y 247.011,Z 618.457,A -85,B 0,C 180,E1 -18803.464,E2 -18803.464} C_VEL
LIN {X 0,Y 246.969,Z 621.633,A -85,B 0,C 180,E1 -18806.736,E2 -18806.736} C_VEL
LIN {X 0,Y 247.024,Z 622.686,A -85,B 0,C 180,E1 -18808.368,E2 -18808.368} C_VEL
LIN {X 0,Y 247.031,Z 623.39,A -85,B 0,C 180,E1 -18809.999,E2 -18809.999} C_VEL
LIN {X 0,Y 247.003,Z 623.752,A -85,B 0,C 180,E1 -18811.629,E2 -18811.629} C_VEL
LIN {X 0,Y 246.883,Z 623.468,A -85,B 0,C 180,E1 -18814.898,E2 -18814.898} C_VEL
LIN {X 0,Y 247.152,Z 621.865,A -85,B 0,C 180,E1 -18818.172,E2 -18818.172} C_VEL
LIN {X 0,Y 247.882,Z 618.919,A -85,B 0,C 180,E1 -18821.446,E2 -18821.446} C_VEL
LIN {X 0,Y 249.322,Z 614.561,A -85,B 0,C 180,E1 -18824.695,E2 -18824.695} C_VEL
LIN {X 0,Y 251.347,Z 608.672,A -85,B 0,C 180,E1 -18827.911,E2 -18827.911} C_VEL
LIN {X 0,Y 253.78,Z 602.094,A -85,B 0,C 180,E1 -18830.675,E2 -18830.675} C_VEL
LIN {X 0,Y 256.861,Z 593.989,A -85,B 0,C 180,E1 -18833.373,E2 -18833.373} C_VEL
LIN {X 0,Y 259.98,Z 585.546,A -85,B 0,C 180,E1 -18835.626,E2 -18835.626} C_VEL
LIN {X 0,Y 263.59,Z 575.398,A -85,B 0,C 180,E1 -18837.812,E2 -18837.812} C_VEL
LIN {X 0,Y 266.875,Z 564.908,A -85,B 0,C 180,E1 -18839.652,E2 -18839.652} C_VEL
LIN {X 0,Y 270.287,Z 552.909,A -85,B 0,C 180,E1 -18841.333,E2 -18841.333} C_VEL
LIN {X 0,Y 273.336,Z 540.735,A -85,B 0,C 180,E1 -18842.678,E2 -18842.678} C_VEL
LIN {X 0,Y 276.22,Z 527.231,A -85,B 0,C 180,E1 -18843.817,E2 -18843.817} C_VEL
LIN {X 0,Y 278.533,Z 513.131,A -85,B 0,C 180,E1 -18844.7,E2 -18844.7} C_VEL
LIN {X 0,Y 280.223,Z 498.794,A -85,B 0,C 180,E1 -18845.307,E2 -18845.307} C_VEL
LIN {X 0,Y 282.187,Z 462.013,A -85,B 0,C 180,E1 -18846.281,E2 -18846.281} C_VEL
LIN {X 0,Y 284.21,Z 420.821,A -85,B 0,C 180,E1 -18847.332,E2 -18847.332} C_VEL
LIN {X 0,Y 282.967,Z 412.754,A -85,B 0,C 180,E1 -18847.853,E2 -18847.853} C_VEL
LIN {X 0,Y 276.213,Z 397.773,A -85,B 0,C 180,E1 -18849.77,E2 -18849.77} C_VEL
LIN {X 0,Y 268.964,Z 384.107,A -85,B 0,C 180,E1 -18851.915,E2 -18851.915} C_VEL
LIN {X 0,Y 262.526,Z 373.417,A -85,B 0,C 180,E1 -18853.954,E2 -18853.954} C_VEL
LIN {X 0,Y 259.354,Z 368.453,A -85,B 0,C 180,E1 -18855.023,E2 -18855.023} C_VEL
LIN {X 0,Y 255.462,Z 362.603,A -85,B 0,C 180,E1 -18856.409,E2 -18856.409} C_VEL
LIN {X 0,Y 252.412,Z 358.07,A -85,B 0,C 180,E1 -18857.558,E2 -18857.558} C_VEL
LIN {X 0,Y 252.135,Z 357.481,A -85,B 0,C 180,E1 -18857.698,E2 -18857.698} C_VEL
LIN {X 0,Y 249.921,Z 350.639,A -85,B 0,C 180,E1 -18861.781,E2 -18861.781} C_VEL
LIN {X 0,Y 249.065,Z 348.082,A -85,B 0,C 180,E1 -18863.494,E2 -18863.494} C_VEL
LIN {X 0,Y 249.035,Z 348.083,A -85,B 0,C 180,E1 -18867.843,E2 -18867.843} C_VEL
LIN {X 0,Y 249.092,Z 348.078,A -85,B 0,C 180,E1 -18871.337,E2 -18871.337} C_VEL
LIN {X 0,Y 249.146,Z 348.074,A -85,B 0,C 180,E1 -18874.967,E2 -18874.967} C_VEL
LIN {X 0,Y 249.104,Z 348.072,A -85,B 0,C 180,E1 -18880.21,E2 -18880.21} C_VEL
LIN {X 0,Y 249.236,Z 348.06,A -85,B 0,C 180,E1 -18883.621,E2 -18883.621} C_VEL
LIN {X 0,Y 249.246,Z 348.051,A -85,B 0,C 180,E1 -18888.616,E2 -18888.616} C_VEL
LIN {X 0,Y 249.477,Z 348.028,A -85,B 0,C 180,E1 -18891.902,E2 -18891.902} C_VEL
LIN {X 0,Y 249.274,Z 348.06,A -85,B 0,C 180,E1 -18895.147,E2 -18895.147} C_VEL
LIN {X 0,Y 249.655,Z 348.006,A -85,B 0,C 180,E1 -18898.386,E2 -18898.386} C_VEL
LIN {X 0,Y 249.65,Z 348.001,A -85,B 0,C 180,E1 -18901.613,E2 -18901.613} C_VEL
LIN {X 0,Y 249.412,Z 348.037,A -85,B 0,C 180,E1 -18906.543,E2 -18906.543} C_VEL
LIN {X 0,Y 249.334,Z 348.043,A -85,B 0,C 180,E1 -18909.736,E2 -18909.736} C_VEL
LIN {X 0,Y 249.163,Z 348.074,A -85,B 0,C 180,E1 -18914.705,E2 -18914.705} C_VEL
LIN {X 0,Y 249.094,Z 348.082,A -85,B 0,C 180,E1 -18918.08,E2 -18918.08} C_VEL
LIN {X 0,Y 249.072,Z 348.081,A -85,B 0,C 180,E1 -18921.519,E2 -18921.519} C_VEL
LIN {X 0,Y 249.046,Z 348.087,A -85,B 0,C 180,E1 -18923.38,E2 -18923.38} C_VEL
LIN {X 0,Y 249.834,Z 350.572,A -85,B 0,C 180,E1 -18923.796,E2 -18923.796} C_VEL
LIN {X 0,Y 251.989,Z 352.977,A -85,B 0,C 180,E1 -18924.62,E2 -18924.62} C_VEL
LIN {X 0,Y 252.971,Z 353.742,A -85,B 0,C 180,E1 -18924.968,E2 -18924.968} C_VEL
LIN {X 0,Y 254.976,Z 357.043,A -85,B 0,C 180,E1 -18925.743,E2 -18925.743} C_VEL
LIN {X 0,Y 256.983,Z 359.173,A -85,B 0,C 180,E1 -18926.439,E2 -18926.439} C_VEL
LIN {X 0,Y 259.472,Z 362.577,A -85,B 0,C 180,E1 -18927.307,E2 -18927.307} C_VEL
LIN {X 0,Y 266.647,Z 372.52,A -85,B 0,C 180,E1 -18929.623,E2 -18929.623} C_VEL
LIN {X 0,Y 271.561,Z 380.052,A -85,B 0,C 180,E1 -18931.089,E2 -18931.089} C_VEL
LIN {X 0,Y 277.609,Z 390.733,A -85,B 0,C 180,E1 -18932.828,E2 -18932.828} C_VEL
LIN {X 0,Y 284.157,Z 403.927,A -85,B 0,C 180,E1 -18934.629,E2 -18934.629} C_VEL
LIN {X 0,Y 285.018,Z 405.782,A -85,B 0,C 180,E1 -18934.86,E2 -18934.86} C_VEL
LIN {X 0,Y 280.987,Z 481.548,A -85,B 0,C 180,E1 -18936.786,E2 -18936.786} C_VEL
LIN {X 0,Y 279.539,Z 495.996,A -85,B 0,C 180,E1 -18937.418,E2 -18937.418} C_VEL
LIN {X 0,Y 277.524,Z 509.602,A -85,B 0,C 180,E1 -18938.278,E2 -18938.278} C_VEL
LIN {X 0,Y 275.162,Z 522.657,A -85,B 0,C 180,E1 -18939.412,E2 -18939.412} C_VEL
LIN {X 0,Y 272.425,Z 534.628,A -85,B 0,C 180,E1 -18940.731,E2 -18940.731} C_VEL
LIN {X 0,Y 269.412,Z 545.758,A -85,B 0,C 180,E1 -18942.254,E2 -18942.254} C_VEL
LIN {X 0,Y 265.886,Z 557.196,A -85,B 0,C 180,E1 -18944.203,E2 -18944.203} C_VEL
LIN {X 0,Y 262.307,Z 567.771,A -85,B 0,C 180,E1 -18946.468,E2 -18946.468} C_VEL
LIN {X 0,Y 258.991,Z 576.682,A -85,B 0,C 180,E1 -18948.851,E2 -18948.851} C_VEL
LIN {X 0,Y 256.021,Z 584.196,A -85,B 0,C 180,E1 -18951.356,E2 -18951.356} C_VEL
LIN {X 0,Y 253.136,Z 591.202,A -85,B 0,C 180,E1 -18954.338,E2 -18954.338} C_VEL
LIN {X 0,Y 251.045,Z 596.259,A -85,B 0,C 180,E1 -18957.123,E2 -18957.123} C_VEL
LIN {X 0,Y 249.612,Z 599.647,A -85,B 0,C 180,E1 -18959.551,E2 -18959.551} C_VEL
LIN {X 0,Y 248.796,Z 601.58,A -85,B 0,C 180,E1 -18961.302,E2 -18961.302} C_VEL
LIN {X 0,Y 248.111,Z 603.084,A -85,B 0,C 180,E1 -18963.052,E2 -18963.052} C_VEL
LIN {X 0,Y 247.204,Z 604.902,A -85,B 0,C 180,E1 -18966.547,E2 -18966.547} C_VEL
LIN {X 0,Y 246.747,Z 605.237,A -85,B 0,C 180,E1 -18970.037,E2 -18970.037} C_VEL
LIN {X 0,Y 246.663,Z 604.138,A -85,B 0,C 180,E1 -18973.447,E2 -18973.447} C_VEL
LIN {X 0,Y 246.79,Z 602.789,A -85,B 0,C 180,E1 -18975.518,E2 -18975.518} C_VEL
LIN {X 0,Y 247.181,Z 599.802,A -85,B 0,C 180,E1 -18978.521,E2 -18978.521} C_VEL
LIN {X 0,Y 247.728,Z 596.33,A -85,B 0,C 180,E1 -18981.025,E2 -18981.025} C_VEL
LIN {X 0,Y 248.525,Z 591.971,A -85,B 0,C 180,E1 -18983.507,E2 -18983.507} C_VEL
LIN {X 0,Y 249.678,Z 585.628,A -85,B 0,C 180,E1 -18986.37,E2 -18986.37} C_VEL
LIN {X 0,Y 251.332,Z 577.717,A -85,B 0,C 180,E1 -18989.2,E2 -18989.2} C_VEL
LIN {X 0,Y 253.103,Z 569.451,A -85,B 0,C 180,E1 -18991.593,E2 -18991.593} C_VEL
LIN {X 0,Y 255.108,Z 559.514,A -85,B 0,C 180,E1 -18993.951,E2 -18993.951} C_VEL
LIN {X 0,Y 257.382,Z 548.431,A -85,B 0,C 180,E1 -18996.075,E2 -18996.075} C_VEL
LIN {X 0,Y 259.62,Z 536.081,A -85,B 0,C 180,E1 -18997.976,E2 -18997.976} C_VEL
LIN {X 0,Y 261.638,Z 523.81,A -85,B 0,C 180,E1 -18999.471,E2 -18999.471} C_VEL
LIN {X 0,Y 263.494,Z 510.201,A -85,B 0,C 180,E1 -19000.762,E2 -19000.762} C_VEL
LIN {X 0,Y 264.897,Z 496.02,A -85,B 0,C 180,E1 -19001.77,E2 -19001.77} C_VEL
LIN {X 0,Y 266.015,Z 481.4,A -85,B 0,C 180,E1 -19002.469,E2 -19002.469} C_VEL
LIN {X 0,Y 267.353,Z 447.894,A -85,B 0,C 180,E1 -19003.393,E2 -19003.393} C_VEL
LIN {X 0,Y 269.356,Z 392.613,A -85,B 0,C 180,E1 -19004.843,E2 -19004.843} C_VEL
LIN {X 0,Y 261.847,Z 373.568,A -85,B 0,C 180,E1 -19006.302,E2 -19006.302} C_VEL
LIN {X 0,Y 256.756,Z 363.003,A -85,B 0,C 180,E1 -19007.272,E2 -19007.272} C_VEL
LIN {X 0,Y 250.129,Z 350.941,A -85,B 0,C 180,E1 -19008.546,E2 -19008.546} C_VEL
LIN {X 0,Y 249.108,Z 348.087,A -85,B 0,C 180,E1 -19008.828,E2 -19008.828} C_VEL
LIN {X 0,Y 249.053,Z 348.09,A -85,B 0,C 180,E1 -19013.271,E2 -19013.271} C_VEL
LIN {X 0,Y 249.029,Z 348.091,A -85,B 0,C 180,E1 -19016.844,E2 -19016.844} C_VEL
LIN {X 0,Y 248.994,Z 348.095,A -85,B 0,C 180,E1 -19020.536,E2 -19020.536} C_VEL
LIN {X 0,Y 249.043,Z 348.089,A -85,B 0,C 180,E1 -19024.362,E2 -19024.362} C_VEL
LIN {X 0,Y 249.022,Z 348.085,A -85,B 0,C 180,E1 -19028.383,E2 -19028.383} C_VEL
LIN {X 0,Y 248.97,Z 348.086,A -85,B 0,C 180,E1 -19032.784,E2 -19032.784} C_VEL
LIN {X 0,Y 248.978,Z 348.093,A -85,B 0,C 180,E1 -19037.356,E2 -19037.356} C_VEL
LIN {X 0,Y 249.022,Z 348.075,A -85,B 0,C 180,E1 -19042.208,E2 -19042.208} C_VEL
LIN {X 0,Y 249.044,Z 348.073,A -85,B 0,C 180,E1 -19045.64,E2 -19045.64} C_VEL
LIN {X 0,Y 248.996,Z 348.092,A -85,B 0,C 180,E1 -19049.466,E2 -19049.466} C_VEL
LIN {X 0,Y 249.015,Z 348.087,A -85,B 0,C 180,E1 -19053.156,E2 -19053.156} C_VEL
LIN {X 0,Y 249.008,Z 348.089,A -85,B 0,C 180,E1 -19056.726,E2 -19056.726} C_VEL
LIN {X 0,Y 249.047,Z 348.086,A -85,B 0,C 180,E1 -19060.207,E2 -19060.207} C_VEL
LIN {X 0,Y 249.161,Z 348.069,A -85,B 0,C 180,E1 -19063.617,E2 -19063.617} C_VEL
LIN {X 0,Y 249.222,Z 348.041,A -85,B 0,C 180,E1 -19068.616,E2 -19068.616} C_VEL
LIN {X 0,Y 249.419,Z 348.037,A -85,B 0,C 180,E1 -19071.901,E2 -19071.901} C_VEL
LIN {X 0,Y 249.277,Z 348.055,A -85,B 0,C 180,E1 -19075.149,E2 -19075.149} C_VEL
LIN {X 0,Y 249.67,Z 347.986,A -85,B 0,C 180,E1 -19078.388,E2 -19078.388} C_VEL
LIN {X 0,Y 249.664,Z 347.986,A -85,B 0,C 180,E1 -19080.834,E2 -19080.834} C_VEL
LIN {X 0,Y 248.952,Z 348.088,A -85,B 0,C 180,E1 -19082.176,E2 -19082.176} C_VEL
LIN {X 0,Y 245.989,Z 348.468,A -85,B 0,C 180,E1 -19084.361,E2 -19084.361} C_VEL
LIN {X 0,Y 243.498,Z 348.778,A -85,B 0,C 180,E1 -19086.141,E2 -19086.141} C_VEL
LIN {X 0,Y 242.453,Z 348.906,A -85,B 0,C 180,E1 -19087.525,E2 -19087.525} C_VEL
LIN {X 0,Y 242.38,Z 348.91,A -85,B 0,C 180,E1 -19087.995,E2 -19087.995} C_VEL
LIN {X 0,Y 242.181,Z 348.944,A -85,B 0,C 180,E1 -19091.721,E2 -19091.721} C_VEL
LIN {X 0,Y 242.169,Z 348.943,A -85,B 0,C 180,E1 -19096.722,E2 -19096.722} C_VEL
LIN {X 0,Y 242.059,Z 348.957,A -85,B 0,C 180,E1 -19101.703,E2 -19101.703} C_VEL
LIN {X 0,Y 242.072,Z 348.951,A -85,B 0,C 180,E1 -19105.838,E2 -19105.838} C_VEL
LIN {X 0,Y 242.013,Z 348.958,A -85,B 0,C 180,E1 -19109.583,E2 -19109.583} C_VEL
LIN {X 0,Y 241.986,Z 348.964,A -85,B 0,C 180,E1 -19113.492,E2 -19113.492} C_VEL
LIN {X 0,Y 241.994,Z 348.955,A -85,B 0,C 180,E1 -19117.582,E2 -19117.582} C_VEL
LIN {X 0,Y 241.944,Z 348.972,A -85,B 0,C 180,E1 -19121.922,E2 -19121.922} C_VEL
LIN {X 0,Y 241.942,Z 348.966,A -85,B 0,C 180,E1 -19126.57,E2 -19126.57} C_VEL
LIN {X 0,Y 241.978,Z 348.982,A -85,B 0,C 180,E1 -19128.354,E2 -19128.354} C_VEL
LIN {X 0,Y 244.685,Z 359.71,A -85,B 0,C 180,E1 -19132.465,E2 -19132.465} C_VEL
LIN {X 0,Y 253.795,Z 380.776,A -85,B 0,C 180,E1 -19134.399,E2 -19134.399} C_VEL
LIN {X 0,Y 259.35,Z 395.638,A -85,B 0,C 180,E1 -19135.565,E2 -19135.565} C_VEL
LIN {X 0,Y 262.373,Z 419.063,A -85,B 0,C 180,E1 -19136.651,E2 -19136.651} C_VEL
LIN {X 0,Y 259.244,Z 498.849,A -85,B 0,C 180,E1 -19138.826,E2 -19138.826} C_VEL
LIN {X 0,Y 258.035,Z 513.356,A -85,B 0,C 180,E1 -19139.516,E2 -19139.516} C_VEL
LIN {X 0,Y 256.468,Z 526.751,A -85,B 0,C 180,E1 -19140.444,E2 -19140.444} C_VEL
LIN {X 0,Y 254.625,Z 538.992,A -85,B 0,C 180,E1 -19141.566,E2 -19141.566} C_VEL
LIN {X 0,Y 252.38,Z 552.168,A -85,B 0,C 180,E1 -19143.134,E2 -19143.134} C_VEL
LIN {X 0,Y 250.592,Z 561.256,A -85,B 0,C 180,E1 -19144.455,E2 -19144.455} C_VEL
LIN {X 0,Y 248.543,Z 571.422,A -85,B 0,C 180,E1 -19146.236,E2 -19146.236} C_VEL
LIN {X 0,Y 246.462,Z 580.889,A -85,B 0,C 180,E1 -19148.24,E2 -19148.24} C_VEL
LIN {X 0,Y 244.416,Z 590.376,A -85,B 0,C 180,E1 -19150.689,E2 -19150.689} C_VEL
LIN {X 0,Y 242.791,Z 598.249,A -85,B 0,C 180,E1 -19153.173,E2 -19153.173} C_VEL
LIN {X 0,Y 241.654,Z 604.779,A -85,B 0,C 180,E1 -19155.686,E2 -19155.686} C_VEL
LIN {X 0,Y 240.661,Z 610.143,A -85,B 0,C 180,E1 -19158.203,E2 -19158.203} C_VEL
LIN {X 0,Y 240.183,Z 614.529,A -85,B 0,C 180,E1 -19160.737,E2 -19160.737} C_VEL
LIN {X 0,Y 239.95,Z 617.999,A -85,B 0,C 180,E1 -19163.27,E2 -19163.27} C_VEL
LIN {X 0,Y 239.868,Z 621.256,A -85,B 0,C 180,E1 -19166.639,E2 -19166.639} C_VEL
LIN {X 0,Y 239.953,Z 622.341,A -85,B 0,C 180,E1 -19168.32,E2 -19168.32} C_VEL
LIN {X 0,Y 239.96,Z 623.076,A -85,B 0,C 180,E1 -19169.998,E2 -19169.998} C_VEL
LIN {X 0,Y 239.908,Z 623.467,A -85,B 0,C 180,E1 -19171.677,E2 -19171.677} C_VEL
LIN {X 0,Y 239.801,Z 623.242,A -85,B 0,C 180,E1 -19175.043,E2 -19175.043} C_VEL
LIN {X 0,Y 240.083,Z 621.699,A -85,B 0,C 180,E1 -19178.415,E2 -19178.415} C_VEL
LIN {X 0,Y 240.865,Z 618.815,A -85,B 0,C 180,E1 -19181.784,E2 -19181.784} C_VEL
LIN {X 0,Y 242.433,Z 614.528,A -85,B 0,C 180,E1 -19185.122,E2 -19185.122} C_VEL
LIN {X 0,Y 244.581,Z 608.555,A -85,B 0,C 180,E1 -19188.512,E2 -19188.512} C_VEL
LIN {X 0,Y 247.554,Z 601.206,A -85,B 0,C 180,E1 -19191.656,E2 -19191.656} C_VEL
LIN {X 0,Y 250.9,Z 592.922,A -85,B 0,C 180,E1 -19194.402,E2 -19194.402} C_VEL
LIN {X 0,Y 254.265,Z 584.33,A -85,B 0,C 180,E1 -19196.688,E2 -19196.688} C_VEL
